LIN {X 0,Y 403.243,Z 462.44,A -85,B 0,C 180,E1 10044.516,E2 10044.516} C_VEL
LIN {X 0,Y 403.34,Z 462.44,A -85,B 0,C 180,E1 10050.792,E2 10050.792} C_VEL
LIN {X 0,Y 403.639,Z 462.44,A -85,B 0,C 180,E1 10057.97,E2 10057.97} C_VEL
LIN {X 0,Y 403.729,Z 462.44,A -85,B 0,C 180,E1 10064.781,E2 10064.781} C_VEL
LIN {X 0,Y 404.101,Z 462.44,A -85,B 0,C 180,E1 10071.38,E2 10071.38} C_VEL
LIN {X 0,Y 404.558,Z 462.44,A -85,B 0,C 180,E1 10077.854,E2 10077.854} C_VEL
LIN {X 0,Y 404.307,Z 462.44,A -85,B 0,C 180,E1 10084.294,E2 10084.294} C_VEL
LIN {X 0,Y 403.998,Z 462.44,A -85,B 0,C 180,E1 10090.798,E2 10090.798} C_VEL
LIN {X 0,Y 403.763,Z 462.44,A -85,B 0,C 180,E1 10097.454,E2 10097.454} C_VEL
LIN {X 0,Y 403.46,Z 462.44,A -85,B 0,C 180,E1 10104.377,E2 10104.377} C_VEL
LIN {X 0,Y 403.325,Z 462.44,A -85,B 0,C 180,E1 10111.701,E2 10111.701} C_VEL
LIN {X 0,Y 403.126,Z 462.44,A -85,B 0,C 180,E1 10117.931,E2 10117.931} C_VEL
LIN {X 0,Y 403.183,Z 462.44,A -85,B 0,C 180,E1 10120.032,E2 10120.032} C_VEL
LIN {X 0,Y 405.626,Z 468.108,A -85,B 0,C 180,E1 10120.64,E2 10120.64} C_VEL
LIN {X 0,Y 425.184,Z 498.302,A -85,B 0,C 180,E1 10124.569,E2 10124.569} C_VEL
LIN {X 0,Y 444.51,Z 533.173,A -85,B 0,C 180,E1 10128.253,E2 10128.253} C_VEL
LIN {X 0,Y 440.339,Z 572.363,A -85,B 0,C 180,E1 10129.774,E2 10129.774} C_VEL
LIN {X 0,Y 434.42,Z 610.186,A -85,B 0,C 180,E1 10132.076,E2 10132.076} C_VEL
LIN {X 0,Y 427.708,Z 644.738,A -85,B 0,C 180,E1 10135.102,E2 10135.102} C_VEL
LIN {X 0,Y 420.828,Z 675.887,A -85,B 0,C 180,E1 10138.855,E2 10138.855} C_VEL
LIN {X 0,Y 414.66,Z 702.51,A -85,B 0,C 180,E1 10143.183,E2 10143.183} C_VEL
LIN {X 0,Y 409.869,Z 724.536,A -85,B 0,C 180,E1 10148.032,E2 10148.032} C_VEL
LIN {X 0,Y 406.864,Z 741.838,A -85,B 0,C 180,E1 10153.237,E2 10153.237} C_VEL
LIN {X 0,Y 405.434,Z 753.406,A -85,B 0,C 180,E1 10158.147,E2 10158.147} C_VEL
LIN {X 0,Y 404.793,Z 761.392,A -85,B 0,C 180,E1 10163.557,E2 10163.557} C_VEL
LIN {X 0,Y 404.608,Z 764.387,A -85,B 0,C 180,E1 10167.855,E2 10167.855} C_VEL
LIN {X 0,Y 404.711,Z 764.342,A -85,B 0,C 180,E1 10172.144,E2 10172.144} C_VEL
LIN {X 0,Y 404.926,Z 759.627,A -85,B 0,C 180,E1 10177.899,E2 10177.899} C_VEL
LIN {X 0,Y 405.887,Z 749.624,A -85,B 0,C 180,E1 10183.577,E2 10183.577} C_VEL
LIN {X 0,Y 407.987,Z 735.102,A -85,B 0,C 180,E1 10188.911,E2 10188.911} C_VEL
LIN {X 0,Y 412.168,Z 713.862,A -85,B 0,C 180,E1 10194.411,E2 10194.411} C_VEL
LIN {X 0,Y 417.696,Z 689.379,A -85,B 0,C 180,E1 10199.022,E2 10199.022} C_VEL
LIN {X 0,Y 424.22,Z 660.818,A -85,B 0,C 180,E1 10203.015,E2 10203.015} C_VEL
LIN {X 0,Y 431.025,Z 628.305,A -85,B 0,C 180,E1 10206.373,E2 10206.373} C_VEL
LIN {X 0,Y 437.479,Z 591.662,A -85,B 0,C 180,E1 10209.075,E2 10209.075} C_VEL
LIN {X 0,Y 442.599,Z 553.853,A -85,B 0,C 180,E1 10210.941,E2 10210.941} C_VEL
LIN {X 0,Y 443.958,Z 532.295,A -85,B 0,C 180,E1 10211.76,E2 10211.76} C_VEL
LIN {X 0,Y 421.037,Z 491.321,A -85,B 0,C 180,E1 10216.122,E2 10216.122} C_VEL
LIN {X 0,Y 405.693,Z 468.193,A -85,B 0,C 180,E1 10219.241,E2 10219.241} C_VEL
LIN {X 0,Y 403.188,Z 463.26,A -85,B 0,C 180,E1 10219.825,E2 10219.825} C_VEL
LIN {X 0,Y 403.085,Z 462.44,A -85,B 0,C 180,E1 10222.077,E2 10222.077} C_VEL
LIN {X 0,Y 403.271,Z 462.44,A -85,B 0,C 180,E1 10228.294,E2 10228.294} C_VEL
LIN {X 0,Y 403.494,Z 462.44,A -85,B 0,C 180,E1 10235.625,E2 10235.625} C_VEL
LIN {X 0,Y 403.856,Z 462.44,A -85,B 0,C 180,E1 10242.55,E2 10242.55} C_VEL
LIN {X 0,Y 404.065,Z 462.44,A -85,B 0,C 180,E1 10249.204,E2 10249.204} C_VEL
LIN {X 0,Y 404.383,Z 462.44,A -85,B 0,C 180,E1 10255.707,E2 10255.707} C_VEL
LIN {X 0,Y 404.56,Z 462.44,A -85,B 0,C 180,E1 10262.146,E2 10262.146} C_VEL
LIN {X 0,Y 404.134,Z 462.44,A -85,B 0,C 180,E1 10268.619,E2 10268.619} C_VEL
LIN {X 0,Y 403.837,Z 462.44,A -85,B 0,C 180,E1 10275.215,E2 10275.215} C_VEL
LIN {X 0,Y 403.621,Z 462.44,A -85,B 0,C 180,E1 10282.031,E2 10282.031} C_VEL
LIN {X 0,Y 403.342,Z 462.44,A -85,B 0,C 180,E1 10289.208,E2 10289.208} C_VEL
LIN {X 0,Y 403.244,Z 462.475,A -85,B 0,C 180,E1 10295.573,E2 10295.573} C_VEL
LIN {X 0,Y 405.552,Z 467.996,A -85,B 0,C 180,E1 10296.151,E2 10296.151} C_VEL
LIN {X 0,Y 424.512,Z 497.638,A -85,B 0,C 180,E1 10300.032,E2 10300.032} C_VEL
LIN {X 0,Y 439.136,Z 526.934,A -85,B 0,C 180,E1 10302.999,E2 10302.999} C_VEL
LIN {X 0,Y 444.863,Z 542.463,A -85,B 0,C 180,E1 10304.377,E2 10304.377} C_VEL
LIN {X 0,Y 439.664,Z 585.502,A -85,B 0,C 180,E1 10306.314,E2 10306.314} C_VEL
LIN {X 0,Y 433.203,Z 625.818,A -85,B 0,C 180,E1 10309.015,E2 10309.015} C_VEL
LIN {X 0,Y 425.789,Z 664.948,A -85,B 0,C 180,E1 10312.666,E2 10312.666} C_VEL
LIN {X 0,Y 418.809,Z 700.533,A -85,B 0,C 180,E1 10317.16,E2 10317.16} C_VEL
LIN {X 0,Y 413.329,Z 728.728,A -85,B 0,C 180,E1 10321.859,E2 10321.859} C_VEL
LIN {X 0,Y 409.238,Z 752.029,A -85,B 0,C 180,E1 10327.011,E2 10327.011} C_VEL
LIN {X 0,Y 408.927,Z 753.833,A -85,B 0,C 180,E1 10327.49,E2 10327.49} C_VEL
LIN {X 0,Y 403.851,Z 761.699,A -85,B 0,C 180,E1 10329.579,E2 10329.579} C_VEL
LIN {X 0,Y 399.002,Z 768.751,A -85,B 0,C 180,E1 10331.769,E2 10331.769} C_VEL
LIN {X 0,Y 397.398,Z 781.94,A -85,B 0,C 180,E1 10337.345,E2 10337.345} C_VEL
LIN {X 0,Y 396.842,Z 790.704,A -85,B 0,C 180,E1 10343.427,E2 10343.427} C_VEL
LIN {X 0,Y 396.811,Z 793.55,A -85,B 0,C 180,E1 10347.813,E2 10347.813} C_VEL
LIN {X 0,Y 396.709,Z 793.546,A -85,B 0,C 180,E1 10352.187,E2 10352.187} C_VEL
LIN {X 0,Y 396.845,Z 789.894,A -85,B 0,C 180,E1 10357.292,E2 10357.292} C_VEL
LIN {X 0,Y 397.495,Z 780.875,A -85,B 0,C 180,E1 10363.212,E2 10363.212} C_VEL
LIN {X 0,Y 399.257,Z 766.259,A -85,B 0,C 180,E1 10369.111,E2 10369.111} C_VEL
LIN {X 0,Y 402.776,Z 744.884,A -85,B 0,C 180,E1 10375.086,E2 10375.086} C_VEL
LIN {X 0,Y 408.167,Z 717.248,A -85,B 0,C 180,E1 10380.668,E2 10380.668} C_VEL
LIN {X 0,Y 415.013,Z 684.684,A -85,B 0,C 180,E1 10385.557,E2 10385.557} C_VEL
LIN {X 0,Y 422.33,Z 649.108,A -85,B 0,C 180,E1 10389.586,E2 10389.586} C_VEL
LIN {X 0,Y 429.644,Z 609.889,A -85,B 0,C 180,E1 10392.846,E2 10392.846} C_VEL
LIN {X 0,Y 436.016,Z 568.538,A -85,B 0,C 180,E1 10395.251,E2 10395.251} C_VEL
LIN {X 0,Y 438.609,Z 543.556,A -85,B 0,C 180,E1 10396.341,E2 10396.341} C_VEL
LIN {X 0,Y 424.38,Z 510.888,A -85,B 0,C 180,E1 10399.602,E2 10399.602} C_VEL
LIN {X 0,Y 405.652,Z 479.832,A -85,B 0,C 180,E1 10403.499,E2 10403.499} C_VEL
LIN {X 0,Y 397.6,Z 467.995,A -85,B 0,C 180,E1 10405.329,E2 10405.329} C_VEL
LIN {X 0,Y 395.292,Z 462.44,A -85,B 0,C 180,E1 10406.071,E2 10406.071} C_VEL
LIN {X 0,Y 395.454,Z 462.44,A -85,B 0,C 180,E1 10412.65,E2 10412.65} C_VEL
LIN {X 0,Y 395.789,Z 462.44,A -85,B 0,C 180,E1 10419.862,E2 10419.862} C_VEL
LIN {X 0,Y 395.862,Z 462.44,A -85,B 0,C 180,E1 10426.733,E2 10426.733} C_VEL
LIN {X 0,Y 396.337,Z 462.44,A -85,B 0,C 180,E1 10433.418,E2 10433.418} C_VEL
LIN {X 0,Y 396.597,Z 462.44,A -85,B 0,C 180,E1 10439.999,E2 10439.999} C_VEL
LIN {X 0,Y 396.285,Z 462.44,A -85,B 0,C 180,E1 10446.58,E2 10446.58} C_VEL
LIN {X 0,Y 395.984,Z 462.44,A -85,B 0,C 180,E1 10453.26,E2 10453.26} C_VEL
LIN {X 0,Y 395.741,Z 462.44,A -85,B 0,C 180,E1 10460.138,E2 10460.138} C_VEL
LIN {X 0,Y 395.426,Z 462.44,A -85,B 0,C 180,E1 10467.35,E2 10467.35} C_VEL
LIN {X 0,Y 395.339,Z 462.44,A -85,B 0,C 180,E1 10472.585,E2 10472.585} C_VEL
LIN {X 0,Y 395.199,Z 462.44,A -85,B 0,C 180,E1 10478.508,E2 10478.508} C_VEL
LIN {X 0,Y 397.442,Z 467.939,A -85,B 0,C 180,E1 10479.116,E2 10479.116} C_VEL
LIN {X 0,Y 405.055,Z 478.925,A -85,B 0,C 180,E1 10480.822,E2 10480.822} C_VEL
LIN {X 0,Y 425.307,Z 511.342,A -85,B 0,C 180,E1 10484.919,E2 10484.919} C_VEL
LIN {X 0,Y 438.604,Z 537.518,A -85,B 0,C 180,E1 10487.683,E2 10487.683} C_VEL
LIN {X 0,Y 434.209,Z 574.487,A -85,B 0,C 180,E1 10489.169,E2 10489.169} C_VEL
LIN {X 0,Y 428.051,Z 611.767,A -85,B 0,C 180,E1 10491.495,E2 10491.495} C_VEL
LIN {X 0,Y 421.059,Z 645.965,A -85,B 0,C 180,E1 10494.552,E2 10494.552} C_VEL
LIN {X 0,Y 413.986,Z 676.406,A -85,B 0,C 180,E1 10498.281,E2 10498.281} C_VEL
LIN {X 0,Y 407.423,Z 703.332,A -85,B 0,C 180,E1 10502.736,E2 10502.736} C_VEL
LIN {X 0,Y 402.422,Z 725.088,A -85,B 0,C 180,E1 10507.603,E2 10507.603} C_VEL
LIN {X 0,Y 399.181,Z 742.302,A -85,B 0,C 180,E1 10512.905,E2 10512.905} C_VEL
LIN {X 0,Y 397.628,Z 753.785,A -85,B 0,C 180,E1 10517.911,E2 10517.911} C_VEL
LIN {X 0,Y 396.907,Z 761.705,A -85,B 0,C 180,E1 10523.428,E2 10523.428} C_VEL
LIN {X 0,Y 396.71,Z 764.677,A -85,B 0,C 180,E1 10527.813,E2 10527.813} C_VEL
LIN {X 0,Y 396.811,Z 764.633,A -85,B 0,C 180,E1 10532.187,E2 10532.187} C_VEL
LIN {X 0,Y 397.004,Z 760.642,A -85,B 0,C 180,E1 10537.487,E2 10537.487} C_VEL
LIN {X 0,Y 397.944,Z 751.414,A -85,B 0,C 180,E1 10543.197,E2 10543.197} C_VEL
LIN {X 0,Y 400.43,Z 735.516,A -85,B 0,C 180,E1 10549.319,E2 10549.319} C_VEL
LIN {X 0,Y 404.835,Z 714.398,A -85,B 0,C 180,E1 10554.883,E2 10554.883} C_VEL
LIN {X 0,Y 410.779,Z 689.583,A -85,B 0,C 180,E1 10559.617,E2 10559.617} C_VEL
LIN {X 0,Y 417.86,Z 659.909,A -85,B 0,C 180,E1 10563.79,E2 10563.79} C_VEL
LIN {X 0,Y 424.831,Z 628.177,A -85,B 0,C 180,E1 10567.074,E2 10567.074} C_VEL
LIN {X 0,Y 431.426,Z 592.294,A -85,B 0,C 180,E1 10569.748,E2 10569.748} C_VEL
LIN {X 0,Y 436.852,Z 554.113,A -85,B 0,C 180,E1 10571.648,E2 10571.648} C_VEL
LIN {X 0,Y 438.104,Z 535.545,A -85,B 0,C 180,E1 10572.372,E2 10572.372} C_VEL
LIN {X 0,Y 417.025,Z 497.141,A -85,B 0,C 180,E1 10576.609,E2 10576.609} C_VEL
LIN {X 0,Y 398.095,Z 468.555,A -85,B 0,C 180,E1 10580.634,E2 10580.634} C_VEL
LIN {X 0,Y 395.27,Z 463.755,A -85,B 0,C 180,E1 10581.317,E2 10581.317} C_VEL
LIN {X 0,Y 395.179,Z 462.44,A -85,B 0,C 180,E1 10581.434,E2 10581.434} C_VEL
LIN {X 0,Y 395.269,Z 462.44,A -85,B 0,C 180,E1 10587.574,E2 10587.574} C_VEL
LIN {X 0,Y 395.439,Z 462.44,A -85,B 0,C 180,E1 10592.651,E2 10592.651} C_VEL
LIN {X 0,Y 395.796,Z 462.44,A -85,B 0,C 180,E1 10599.865,E2 10599.865} C_VEL
LIN {X 0,Y 396.074,Z 462.44,A -85,B 0,C 180,E1 10606.743,E2 10606.743} C_VEL
LIN {X 0,Y 396.308,Z 462.44,A -85,B 0,C 180,E1 10613.42,E2 10613.42} C_VEL
LIN {X 0,Y 396.666,Z 462.44,A -85,B 0,C 180,E1 10620.001,E2 10620.001} C_VEL
LIN {X 0,Y 396.332,Z 462.44,A -85,B 0,C 180,E1 10626.637,E2 10626.637} C_VEL
LIN {X 0,Y 395.991,Z 462.44,A -85,B 0,C 180,E1 10633.263,E2 10633.263} C_VEL
LIN {X 0,Y 395.757,Z 462.44,A -85,B 0,C 180,E1 10640.14,E2 10640.14} C_VEL
LIN {X 0,Y 395.457,Z 462.44,A -85,B 0,C 180,E1 10647.35,E2 10647.35} C_VEL
LIN {X 0,Y 395.333,Z 462.763,A -85,B 0,C 180,E1 10654.086,E2 10654.086} C_VEL
LIN {X 0,Y 397.8,Z 468.188,A -85,B 0,C 180,E1 10654.732,E2 10654.732} C_VEL
LIN {X 0,Y 414.691,Z 494.071,A -85,B 0,C 180,E1 10658.429,E2 10658.429} C_VEL
LIN {X 0,Y 430.735,Z 523.96,A -85,B 0,C 180,E1 10661.779,E2 10661.779} C_VEL
LIN {X 0,Y 438.795,Z 545.274,A -85,B 0,C 180,E1 10663.776,E2 10663.776} C_VEL
LIN {X 0,Y 433.486,Z 586.598,A -85,B 0,C 180,E1 10665.686,E2 10665.686} C_VEL
LIN {X 0,Y 426.751,Z 626.42,A -85,B 0,C 180,E1 10668.397,E2 10668.397} C_VEL
LIN {X 0,Y 419.033,Z 665.305,A -85,B 0,C 180,E1 10672.1,E2 10672.1} C_VEL
LIN {X 0,Y 411.788,Z 699.678,A -85,B 0,C 180,E1 10676.527,E2 10676.527} C_VEL
LIN {X 0,Y 405.725,Z 729.414,A -85,B 0,C 180,E1 10681.587,E2 10681.587} C_VEL
LIN {X 0,Y 401.316,Z 753.319,A -85,B 0,C 180,E1 10687.039,E2 10687.039} C_VEL
LIN {X 0,Y 399.002,Z 768.751,A -85,B 0,C 180,E1 10691.769,E2 10691.769} C_VEL
LIN {X 0,Y 395.882,Z 773.516,A -85,B 0,C 180,E1 10693.479,E2 10693.479} C_VEL
LIN {X 0,Y 389.845,Z 779.624,A -85,B 0,C 180,E1 10696.09,E2 10696.09} C_VEL
LIN {X 0,Y 389.698,Z 780.266,A -85,B 0,C 180,E1 10696.398,E2 10696.398} C_VEL
LIN {X 0,Y 388.936,Z 789.6,A -85,B 0,C 180,E1 10702.571,E2 10702.571} C_VEL
LIN {X 0,Y 388.915,Z 793.26,A -85,B 0,C 180,E1 10707.769,E2 10707.769} C_VEL
LIN {X 0,Y 388.82,Z 793.257,A -85,B 0,C 180,E1 10712.232,E2 10712.232} C_VEL
LIN {X 0,Y 388.951,Z 789.583,A -85,B 0,C 180,E1 10717.441,E2 10717.441} C_VEL
LIN {X 0,Y 389.639,Z 780.512,A -85,B 0,C 180,E1 10723.483,E2 10723.483} C_VEL
LIN {X 0,Y 391.56,Z 765.572,A -85,B 0,C 180,E1 10729.588,E2 10729.588} C_VEL
LIN {X 0,Y 395.241,Z 744.563,A -85,B 0,C 180,E1 10735.522,E2 10735.522} C_VEL
LIN {X 0,Y 400.986,Z 716.49,A -85,B 0,C 180,E1 10741.279,E2 10741.279} C_VEL
LIN {X 0,Y 408.135,Z 684.775,A -85,B 0,C 180,E1 10746.143,E2 10746.143} C_VEL
LIN {X 0,Y 415.777,Z 649.522,A -85,B 0,C 180,E1 10750.208,E2 10750.208} C_VEL
LIN {X 0,Y 423.285,Z 611.364,A -85,B 0,C 180,E1 10753.443,E2 10753.443} C_VEL
LIN {X 0,Y 430.124,Z 569.177,A -85,B 0,C 180,E1 10755.939,E2 10755.939} C_VEL
LIN {X 0,Y 432.454,Z 546.358,A -85,B 0,C 180,E1 10756.977,E2 10756.977} C_VEL
LIN {X 0,Y 419.8,Z 516.142,A -85,B 0,C 180,E1 10760.099,E2 10760.099} C_VEL
LIN {X 0,Y 401.79,Z 485.729,A -85,B 0,C 180,E1 10764.013,E2 10764.013} C_VEL
LIN {X 0,Y 389.978,Z 468.304,A -85,B 0,C 180,E1 10766.833,E2 10766.833} C_VEL
LIN {X 0,Y 387.541,Z 463.879,A -85,B 0,C 180,E1 10767.49,E2 10767.49} C_VEL
LIN {X 0,Y 387.379,Z 462.44,A -85,B 0,C 180,E1 10767.797,E2 10767.797} C_VEL
LIN {X 0,Y 387.575,Z 462.44,A -85,B 0,C 180,E1 10774.551,E2 10774.551} C_VEL
LIN {X 0,Y 387.855,Z 462.44,A -85,B 0,C 180,E1 10781.803,E2 10781.803} C_VEL
LIN {X 0,Y 388.016,Z 462.44,A -85,B 0,C 180,E1 10788.749,E2 10788.749} C_VEL
LIN {X 0,Y 388.477,Z 462.44,A -85,B 0,C 180,E1 10795.528,E2 10795.528} C_VEL
LIN {X 0,Y 388.705,Z 462.44,A -85,B 0,C 180,E1 10799.999,E2 10799.999} C_VEL
LIN {X 0,Y 388.362,Z 462.44,A -85,B 0,C 180,E1 10806.715,E2 10806.715} C_VEL
LIN {X 0,Y 388.056,Z 462.44,A -85,B 0,C 180,E1 10813.536,E2 10813.536} C_VEL
LIN {X 0,Y 387.764,Z 462.44,A -85,B 0,C 180,E1 10820.571,E2 10820.571} C_VEL
LIN {X 0,Y 387.523,Z 462.44,A -85,B 0,C 180,E1 10827.956,E2 10827.956} C_VEL
LIN {X 0,Y 387.352,Z 462.44,A -85,B 0,C 180,E1 10835.891,E2 10835.891} C_VEL
LIN {X 0,Y 387.335,Z 462.608,A -85,B 0,C 180,E1 10836.907,E2 10836.907} C_VEL
LIN {X 0,Y 389.422,Z 467.801,A -85,B 0,C 180,E1 10837.505,E2 10837.505} C_VEL
LIN {X 0,Y 392.445,Z 471.944,A -85,B 0,C 180,E1 10838.246,E2 10838.246} C_VEL
LIN {X 0,Y 408.063,Z 495.276,A -85,B 0,C 180,E1 10841.77,E2 10841.77} C_VEL
LIN {X 0,Y 427.465,Z 529.122,A -85,B 0,C 180,E1 10845.822,E2 10845.822} C_VEL
LIN {X 0,Y 432.724,Z 539.783,A -85,B 0,C 180,E1 10847.006,E2 10847.006} C_VEL
LIN {X 0,Y 427.988,Z 577.783,A -85,B 0,C 180,E1 10848.614,E2 10848.614} C_VEL
LIN {X 0,Y 421.648,Z 613.614,A -85,B 0,C 180,E1 10850.916,E2 10850.916} C_VEL
LIN {X 0,Y 414.438,Z 647.187,A -85,B 0,C 180,E1 10853.986,E2 10853.986} C_VEL
LIN {X 0,Y 407.189,Z 676.889,A -85,B 0,C 180,E1 10857.688,E2 10857.688} C_VEL
LIN {X 0,Y 400.448,Z 703.232,A -85,B 0,C 180,E1 10862.101,E2 10862.101} C_VEL
LIN {X 0,Y 395.121,Z 725.015,A -85,B 0,C 180,E1 10867.019,E2 10867.019} C_VEL
LIN {X 0,Y 391.537,Z 742.753,A -85,B 0,C 180,E1 10872.56,E2 10872.56} C_VEL
LIN {X 0,Y 389.833,Z 754.166,A -85,B 0,C 180,E1 10877.665,E2 10877.665} C_VEL
LIN {X 0,Y 389.041,Z 762.018,A -85,B 0,C 180,E1 10883.295,E2 10883.295} C_VEL
LIN {X 0,Y 388.821,Z 764.968,A -85,B 0,C 180,E1 10887.768,E2 10887.768} C_VEL
LIN {X 0,Y 388.914,Z 764.925,A -85,B 0,C 180,E1 10892.231,E2 10892.231} C_VEL
LIN {X 0,Y 389.125,Z 760.966,A -85,B 0,C 180,E1 10897.64,E2 10897.64} C_VEL
LIN {X 0,Y 390.152,Z 751.813,A -85,B 0,C 180,E1 10903.465,E2 10903.465} C_VEL
LIN {X 0,Y 392.641,Z 737.037,A -85,B 0,C 180,E1 10909.357,E2 10909.357} C_VEL
LIN {X 0,Y 397.259,Z 716.128,A -85,B 0,C 180,E1 10915.089,E2 10915.089} C_VEL
LIN {X 0,Y 403.73,Z 690.395,A -85,B 0,C 180,E1 10920.126,E2 10920.126} C_VEL
LIN {X 0,Y 411.219,Z 660.619,A -85,B 0,C 180,E1 10924.387,E2 10924.387} C_VEL
LIN {X 0,Y 418.595,Z 628.581,A -85,B 0,C 180,E1 10927.747,E2 10927.747} C_VEL
LIN {X 0,Y 425.592,Z 592.054,A -85,B 0,C 180,E1 10930.488,E2 10930.488} C_VEL
LIN {X 0,Y 431.171,Z 554.253,A -85,B 0,C 180,E1 10932.379,E2 10932.379} C_VEL
LIN {X 0,Y 432.208,Z 538.753,A -85,B 0,C 180,E1 10933.013,E2 10933.013} C_VEL
LIN {X 0,Y 412.626,Z 502.339,A -85,B 0,C 180,E1 10937.189,E2 10937.189} C_VEL
LIN {X 0,Y 394.373,Z 474.672,A -85,B 0,C 180,E1 10941.184,E2 10941.184} C_VEL
LIN {X 0,Y 389.32,Z 467.696,A -85,B 0,C 180,E1 10942.409,E2 10942.409} C_VEL
LIN {X 0,Y 387.274,Z 462.44,A -85,B 0,C 180,E1 10943.056,E2 10943.056} C_VEL
LIN {X 0,Y 387.385,Z 462.44,A -85,B 0,C 180,E1 10949.467,E2 10949.467} C_VEL
LIN {X 0,Y 387.694,Z 462.44,A -85,B 0,C 180,E1 10957.016,E2 10957.016} C_VEL
LIN {X 0,Y 388.062,Z 462.44,A -85,B 0,C 180,E1 10964.153,E2 10964.153} C_VEL
LIN {X 0,Y 388.281,Z 462.44,A -85,B 0,C 180,E1 10971.269,E2 10971.269} C_VEL
LIN {X 0,Y 388.681,Z 462.44,A -85,B 0,C 180,E1 10977.769,E2 10977.769} C_VEL
LIN {X 0,Y 388.48,Z 462.44,A -85,B 0,C 180,E1 10984.472,E2 10984.472} C_VEL
LIN {X 0,Y 388.121,Z 462.44,A -85,B 0,C 180,E1 10991.248,E2 10991.248} C_VEL
LIN {X 0,Y 387.863,Z 462.44,A -85,B 0,C 180,E1 10998.197,E2 10998.197} C_VEL
LIN {X 0,Y 387.577,Z 462.44,A -85,B 0,C 180,E1 11005.449,E2 11005.449} C_VEL
LIN {X 0,Y 387.407,Z 462.44,A -85,B 0,C 180,E1 11012.442,E2 11012.442} C_VEL
LIN {X 0,Y 389.657,Z 467.996,A -85,B 0,C 180,E1 11013.109,E2 11013.109} C_VEL
LIN {X 0,Y 392.574,Z 472.095,A -85,B 0,C 180,E1 11013.835,E2 11013.835} C_VEL
LIN {X 0,Y 409.993,Z 498.604,A -85,B 0,C 180,E1 11017.79,E2 11017.79} C_VEL
LIN {X 0,Y 425.494,Z 528.178,A -85,B 0,C 180,E1 11021.212,E2 11021.212} C_VEL
LIN {X 0,Y 432.694,Z 548.803,A -85,B 0,C 180,E1 11023.191,E2 11023.191} C_VEL
LIN {X 0,Y 427.359,Z 587.739,A -85,B 0,C 180,E1 11025.044,E2 11025.044} C_VEL
LIN {X 0,Y 420.354,Z 627.093,A -85,B 0,C 180,E1 11027.769,E2 11027.769} C_VEL
LIN {X 0,Y 412.507,Z 664.691,A -85,B 0,C 180,E1 11031.391,E2 11031.391} C_VEL
LIN {X 0,Y 404.825,Z 699.054,A -85,B 0,C 180,E1 11035.873,E2 11035.873} C_VEL
LIN {X 0,Y 398.384,Z 728.808,A -85,B 0,C 180,E1 11041.039,E2 11041.039} C_VEL
LIN {X 0,Y 393.818,Z 752.47,A -85,B 0,C 180,E1 11046.491,E2 11046.491} C_VEL
LIN {X 0,Y 390.779,Z 771.449,A -85,B 0,C 180,E1 11052.525,E2 11052.525} C_VEL
LIN {X 0,Y 389.698,Z 780.266,A -85,B 0,C 180,E1 11056.398,E2 11056.398} C_VEL
LIN {X 0,Y 386.9,Z 783.741,A -85,B 0,C 180,E1 11058.22,E2 11058.22} C_VEL
LIN {X 0,Y 381.229,Z 787.741,A -85,B 0,C 180,E1 11061.005,E2 11061.005} C_VEL
LIN {X 0,Y 381.102,Z 788.082,A -85,B 0,C 180,E1 11061.332,E2 11061.332} C_VEL
LIN {X 0,Y 380.951,Z 791.891,A -85,B 0,C 180,E1 11065.441,E2 11065.441} C_VEL
LIN {X 0,Y 381.01,Z 793.329,A -85,B 0,C 180,E1 11070,E2 11070} C_VEL
LIN {X 0,Y 380.927,Z 791.891,A -85,B 0,C 180,E1 11074.56,E2 11074.56} C_VEL
LIN {X 0,Y 381.299,Z 785.926,A -85,B 0,C 180,E1 11080.294,E2 11080.294} C_VEL
LIN {X 0,Y 382.408,Z 775.209,A -85,B 0,C 180,E1 11086.091,E2 11086.091} C_VEL
LIN {X 0,Y 385.045,Z 758.047,A -85,B 0,C 180,E1 11092.242,E2 11092.242} C_VEL
LIN {X 0,Y 389.739,Z 734.384,A -85,B 0,C 180,E1 11098.249,E2 11098.249} C_VEL
LIN {X 0,Y 396.366,Z 705.806,A -85,B 0,C 180,E1 11103.635,E2 11103.635} C_VEL
LIN {X 0,Y 403.963,Z 673.635,A -85,B 0,C 180,E1 11108.205,E2 11108.205} C_VEL
LIN {X 0,Y 412.054,Z 637.549,A -85,B 0,C 180,E1 11112.028,E2 11112.028} C_VEL
LIN {X 0,Y 419.82,Z 597.766,A -85,B 0,C 180,E1 11115.077,E2 11115.077} C_VEL
LIN {X 0,Y 426.104,Z 556.005,A -85,B 0,C 180,E1 11117.286,E2 11117.286} C_VEL
LIN {X 0,Y 426.333,Z 548.846,A -85,B 0,C 180,E1 11117.653,E2 11117.653} C_VEL
LIN {X 0,Y 414.639,Z 520.428,A -85,B 0,C 180,E1 11120.714,E2 11120.714} C_VEL
LIN {X 0,Y 397.507,Z 490.866,A -85,B 0,C 180,E1 11124.646,E2 11124.646} C_VEL
LIN {X 0,Y 382.488,Z 468.624,A -85,B 0,C 180,E1 11128.429,E2 11128.429} C_VEL
LIN {X 0,Y 379.581,Z 463.619,A -85,B 0,C 180,E1 11129.267,E2 11129.267} C_VEL
LIN {X 0,Y 379.525,Z 462.44,A -85,B 0,C 180,E1 11129.428,E2 11129.428} C_VEL
LIN {X 0,Y 379.739,Z 462.44,A -85,B 0,C 180,E1 11136.503,E2 11136.503} C_VEL
LIN {X 0,Y 379.949,Z 462.44,A -85,B 0,C 180,E1 11143.803,E2 11143.803} C_VEL
LIN {X 0,Y 380.3,Z 462.44,A -85,B 0,C 180,E1 11150.836,E2 11150.836} C_VEL
LIN {X 0,Y 380.833,Z 462.44,A -85,B 0,C 180,E1 11157.72,E2 11157.72} C_VEL
LIN {X 0,Y 380.571,Z 462.44,A -85,B 0,C 180,E1 11164.562,E2 11164.562} C_VEL
LIN {X 0,Y 380.2,Z 462.44,A -85,B 0,C 180,E1 11171.483,E2 11171.483} C_VEL
LIN {X 0,Y 379.922,Z 462.44,A -85,B 0,C 180,E1 11178.589,E2 11178.589} C_VEL
LIN {X 0,Y 379.626,Z 462.44,A -85,B 0,C 180,E1 11186.018,E2 11186.018} C_VEL
LIN {X 0,Y 379.443,Z 462.44,A -85,B 0,C 180,E1 11193.957,E2 11193.957} C_VEL
LIN {X 0,Y 379.502,Z 463.265,A -85,B 0,C 180,E1 11195.176,E2 11195.176} C_VEL
LIN {X 0,Y 382.246,Z 468.462,A -85,B 0,C 180,E1 11195.972,E2 11195.972} C_VEL
LIN {X 0,Y 397.826,Z 491.087,A -85,B 0,C 180,E1 11199.829,E2 11199.829} C_VEL
LIN {X 0,Y 417.024,Z 523.235,A -85,B 0,C 180,E1 11204.061,E2 11204.061} C_VEL
LIN {X 0,Y 426.858,Z 543.914,A -85,B 0,C 180,E1 11206.388,E2 11206.388} C_VEL
LIN {X 0,Y 421.449,Z 583.428,A -85,B 0,C 180,E1 11208.172,E2 11208.172} C_VEL
LIN {X 0,Y 414.23,Z 620.638,A -85,B 0,C 180,E1 11210.735,E2 11210.735} C_VEL
LIN {X 0,Y 406.113,Z 655.513,A -85,B 0,C 180,E1 11214.205,E2 11214.205} C_VEL
LIN {X 0,Y 398.416,Z 684.842,A -85,B 0,C 180,E1 11218.21,E2 11218.21} C_VEL
LIN {X 0,Y 391.508,Z 710.43,A -85,B 0,C 180,E1 11222.943,E2 11222.943} C_VEL
LIN {X 0,Y 386.391,Z 731.07,A -85,B 0,C 180,E1 11228.144,E2 11228.144} C_VEL
LIN {X 0,Y 383.093,Z 747.449,A -85,B 0,C 180,E1 11233.939,E2 11233.939} C_VEL
LIN {X 0,Y 381.598,Z 758.283,A -85,B 0,C 180,E1 11239.714,E2 11239.714} C_VEL
LIN {X 0,Y 380.961,Z 764.161,A -85,B 0,C 180,E1 11245.441,E2 11245.441} C_VEL
LIN {X 0,Y 381.01,Z 765.618,A -85,B 0,C 180,E1 11250,E2 11250} C_VEL
LIN {X 0,Y 380.978,Z 764.097,A -85,B 0,C 180,E1 11254.559,E2 11254.559} C_VEL
LIN {X 0,Y 381.612,Z 758.146,A -85,B 0,C 180,E1 11260.285,E2 11260.285} C_VEL
LIN {X 0,Y 383.107,Z 747.252,A -85,B 0,C 180,E1 11266.061,E2 11266.061} C_VEL
LIN {X 0,Y 386.707,Z 729.786,A -85,B 0,C 180,E1 11272.14,E2 11272.14} C_VEL
LIN {X 0,Y 392.328,Z 707.456,A -85,B 0,C 180,E1 11277.589,E2 11277.589} C_VEL
LIN {X 0,Y 399.586,Z 680.53,A -85,B 0,C 180,E1 11282.36,E2 11282.36} C_VEL
LIN {X 0,Y 407.429,Z 650.088,A -85,B 0,C 180,E1 11286.319,E2 11286.319} C_VEL
LIN {X 0,Y 415.129,Z 616.507,A -85,B 0,C 180,E1 11289.494,E2 11289.494} C_VEL
LIN {X 0,Y 421.745,Z 580.922,A -85,B 0,C 180,E1 11291.878,E2 11291.878} C_VEL
LIN {X 0,Y 426.484,Z 542.229,A -85,B 0,C 180,E1 11293.643,E2 11293.643} C_VEL
LIN {X 0,Y 407.388,Z 506.122,A -85,B 0,C 180,E1 11297.956,E2 11297.956} C_VEL
LIN {X 0,Y 390.546,Z 480.485,A -85,B 0,C 180,E1 11301.781,E2 11301.781} C_VEL
LIN {X 0,Y 382.29,Z 468.546,A -85,B 0,C 180,E1 11303.903,E2 11303.903} C_VEL
LIN {X 0,Y 379.426,Z 463.324,A -85,B 0,C 180,E1 11304.724,E2 11304.724} C_VEL
LIN {X 0,Y 379.42,Z 462.44,A -85,B 0,C 180,E1 11305.2,E2 11305.2} C_VEL
LIN {X 0,Y 379.529,Z 462.44,A -85,B 0,C 180,E1 11311.402,E2 11311.402} C_VEL
LIN {X 0,Y 379.851,Z 462.44,A -85,B 0,C 180,E1 11318.98,E2 11318.98} C_VEL
LIN {X 0,Y 380.187,Z 462.44,A -85,B 0,C 180,E1 11326.178,E2 11326.178} C_VEL
LIN {X 0,Y 380.489,Z 462.44,A -85,B 0,C 180,E1 11333.146,E2 11333.146} C_VEL
LIN {X 0,Y 380.869,Z 462.44,A -85,B 0,C 180,E1 11340.001,E2 11340.001} C_VEL
LIN {X 0,Y 380.536,Z 462.44,A -85,B 0,C 180,E1 11346.856,E2 11346.856} C_VEL
LIN {X 0,Y 380.116,Z 462.44,A -85,B 0,C 180,E1 11353.827,E2 11353.827} C_VEL
LIN {X 0,Y 379.841,Z 462.44,A -85,B 0,C 180,E1 11361.023,E2 11361.023} C_VEL
LIN {X 0,Y 379.547,Z 462.44,A -85,B 0,C 180,E1 11368.64,E2 11368.64} C_VEL
LIN {X 0,Y 379.55,Z 463.245,A -85,B 0,C 180,E1 11370.736,E2 11370.736} C_VEL
LIN {X 0,Y 382.238,Z 468.448,A -85,B 0,C 180,E1 11371.532,E2 11371.532} C_VEL
LIN {X 0,Y 396.752,Z 489.652,A -85,B 0,C 180,E1 11375.192,E2 11375.192} C_VEL
LIN {X 0,Y 414.36,Z 519.858,A -85,B 0,C 180,E1 11379.229,E2 11379.229} C_VEL
LIN {X 0,Y 425.95,Z 547.76,A -85,B 0,C 180,E1 11382.24,E2 11382.24} C_VEL
LIN {X 0,Y 426.529,Z 552.791,A -85,B 0,C 180,E1 11382.598,E2 11382.598} C_VEL
LIN {X 0,Y 420.808,Z 591.846,A -85,B 0,C 180,E1 11384.564,E2 11384.564} C_VEL
LIN {X 0,Y 413.84,Z 628.638,A -85,B 0,C 180,E1 11387.195,E2 11387.195} C_VEL
LIN {X 0,Y 405.689,Z 665.745,A -85,B 0,C 180,E1 11390.854,E2 11390.854} C_VEL
LIN {X 0,Y 397.99,Z 698.52,A -85,B 0,C 180,E1 11395.203,E2 11395.203} C_VEL
LIN {X 0,Y 391.14,Z 728.204,A -85,B 0,C 180,E1 11400.45,E2 11400.45} C_VEL
LIN {X 0,Y 386.04,Z 752.939,A -85,B 0,C 180,E1 11406.295,E2 11406.295} C_VEL
LIN {X 0,Y 383.048,Z 771.011,A -85,B 0,C 180,E1 11412.161,E2 11412.161} C_VEL
LIN {X 0,Y 381.39,Z 784.243,A -85,B 0,C 180,E1 11418.551,E2 11418.551} C_VEL
LIN {X 0,Y 381.102,Z 788.082,A -85,B 0,C 180,E1 11421.332,E2 11421.332} C_VEL
LIN {X 0,Y 378.45,Z 790.116,A -85,B 0,C 180,E1 11423.243,E2 11423.243} C_VEL
LIN {X 0,Y 373.102,Z 791.981,A -85,B 0,C 180,E1 11426.138,E2 11426.138} C_VEL
LIN {X 0,Y 373.013,Z 792.122,A -85,B 0,C 180,E1 11426.475,E2 11426.475} C_VEL
LIN {X 0,Y 373.138,Z 793.043,A -85,B 0,C 180,E1 11430,E2 11430} C_VEL
LIN {X 0,Y 373.052,Z 791.595,A -85,B 0,C 180,E1 11434.656,E2 11434.656} C_VEL
LIN {X 0,Y 373.421,Z 785.585,A -85,B 0,C 180,E1 11440.513,E2 11440.513} C_VEL
LIN {X 0,Y 374.604,Z 774.789,A -85,B 0,C 180,E1 11446.436,E2 11446.436} C_VEL
LIN {X 0,Y 377.445,Z 757.567,A -85,B 0,C 180,E1 11452.696,E2 11452.696} C_VEL
LIN {X 0,Y 382.325,Z 734.436,A -85,B 0,C 180,E1 11458.718,E2 11458.718} C_VEL
LIN {X 0,Y 389.406,Z 705.3,A -85,B 0,C 180,E1 11464.319,E2 11464.319} C_VEL
LIN {X 0,Y 397.527,Z 673.117,A -85,B 0,C 180,E1 11468.935,E2 11468.935} C_VEL
LIN {X 0,Y 405.999,Z 636.88,A -85,B 0,C 180,E1 11472.807,E2 11472.807} C_VEL
LIN {X 0,Y 413.953,Z 597.847,A -85,B 0,C 180,E1 11475.821,E2 11475.821} C_VEL
LIN {X 0,Y 420.609,Z 555.138,A -85,B 0,C 180,E1 11478.085,E2 11478.085} C_VEL
LIN {X 0,Y 419.345,Z 548.587,A -85,B 0,C 180,E1 11478.64,E2 11478.64} C_VEL
LIN {X 0,Y 407.727,Z 521.035,A -85,B 0,C 180,E1 11481.794,E2 11481.794} C_VEL
LIN {X 0,Y 390.692,Z 492.079,A -85,B 0,C 180,E1 11485.923,E2 11485.923} C_VEL
LIN {X 0,Y 378.223,Z 474.046,A -85,B 0,C 180,E1 11489.212,E2 11489.212} C_VEL
LIN {X 0,Y 374.692,Z 468.726,A -85,B 0,C 180,E1 11490.248,E2 11490.248} C_VEL
LIN {X 0,Y 371.735,Z 463.859,A -85,B 0,C 180,E1 11491.168,E2 11491.168} C_VEL
LIN {X 0,Y 371.633,Z 462.44,A -85,B 0,C 180,E1 11491.414,E2 11491.414} C_VEL
LIN {X 0,Y 371.879,Z 462.44,A -85,B 0,C 180,E1 11498.505,E2 11498.505} C_VEL
LIN {X 0,Y 372.069,Z 462.44,A -85,B 0,C 180,E1 11505.868,E2 11505.868} C_VEL
LIN {X 0,Y 372.595,Z 462.44,A -85,B 0,C 180,E1 11512.997,E2 11512.997} C_VEL
LIN {X 0,Y 372.902,Z 462.44,A -85,B 0,C 180,E1 11519.999,E2 11519.999} C_VEL
LIN {X 0,Y 372.524,Z 462.44,A -85,B 0,C 180,E1 11527.002,E2 11527.002} C_VEL
LIN {X 0,Y 372.165,Z 462.44,A -85,B 0,C 180,E1 11534.126,E2 11534.126} C_VEL
LIN {X 0,Y 371.826,Z 462.44,A -85,B 0,C 180,E1 11541.495,E2 11541.495} C_VEL
LIN {X 0,Y 371.639,Z 462.44,A -85,B 0,C 180,E1 11546.621,E2 11546.621} C_VEL
LIN {X 0,Y 371.576,Z 462.686,A -85,B 0,C 180,E1 11553.216,E2 11553.216} C_VEL
LIN {X 0,Y 373.707,Z 467.84,A -85,B 0,C 180,E1 11553.933,E2 11553.933} C_VEL
LIN {X 0,Y 376.458,Z 470.959,A -85,B 0,C 180,E1 11554.708,E2 11554.708} C_VEL
LIN {X 0,Y 396.245,Z 500.094,A -85,B 0,C 180,E1 11559.779,E2 11559.779} C_VEL
LIN {X 0,Y 414.948,Z 533.455,A -85,B 0,C 180,E1 11564.156,E2 11564.156} C_VEL
LIN {X 0,Y 420.993,Z 547.013,A -85,B 0,C 180,E1 11565.725,E2 11565.725} C_VEL
LIN {X 0,Y 415.416,Z 585.253,A -85,B 0,C 180,E1 11567.512,E2 11567.512} C_VEL
LIN {X 0,Y 407.818,Z 622.525,A -85,B 0,C 180,E1 11570.145,E2 11570.145} C_VEL
LIN {X 0,Y 399.662,Z 655.996,A -85,B 0,C 180,E1 11573.535,E2 11573.535} C_VEL
LIN {X 0,Y 391.433,Z 685.898,A -85,B 0,C 180,E1 11577.696,E2 11577.696} C_VEL
LIN {X 0,Y 384.323,Z 710.821,A -85,B 0,C 180,E1 11582.395,E2 11582.395} C_VEL
LIN {X 0,Y 378.886,Z 731.437,A -85,B 0,C 180,E1 11587.688,E2 11587.688} C_VEL
LIN {X 0,Y 375.378,Z 747.794,A -85,B 0,C 180,E1 11593.599,E2 11593.599} C_VEL
LIN {X 0,Y 373.748,Z 758.61,A -85,B 0,C 180,E1 11599.496,E2 11599.496} C_VEL
LIN {X 0,Y 373.088,Z 764.461,A -85,B 0,C 180,E1 11605.344,E2 11605.344} C_VEL
LIN {X 0,Y 373.137,Z 765.904,A -85,B 0,C 180,E1 11610,E2 11610} C_VEL
LIN {X 0,Y 373.104,Z 764.396,A -85,B 0,C 180,E1 11614.656,E2 11614.656} C_VEL
LIN {X 0,Y 373.762,Z 758.479,A -85,B 0,C 180,E1 11620.504,E2 11620.504} C_VEL
LIN {X 0,Y 375.399,Z 747.599,A -85,B 0,C 180,E1 11626.4,E2 11626.4} C_VEL
LIN {X 0,Y 379.246,Z 730.167,A -85,B 0,C 180,E1 11632.599,E2 11632.599} C_VEL
LIN {X 0,Y 385.201,Z 707.866,A -85,B 0,C 180,E1 11638.144,E2 11638.144} C_VEL
LIN {X 0,Y 392.762,Z 681.188,A -85,B 0,C 180,E1 11642.957,E2 11642.957} C_VEL
LIN {X 0,Y 401.014,Z 650.609,A -85,B 0,C 180,E1 11646.996,E2 11646.996} C_VEL
LIN {X 0,Y 409.18,Z 616.564,A -85,B 0,C 180,E1 11650.245,E2 11650.245} C_VEL
LIN {X 0,Y 416.139,Z 580.585,A -85,B 0,C 180,E1 11652.662,E2 11652.662} C_VEL
LIN {X 0,Y 420.6,Z 545.375,A -85,B 0,C 180,E1 11654.326,E2 11654.326} C_VEL
LIN {X 0,Y 402.251,Z 509.921,A -85,B 0,C 180,E1 11658.725,E2 11658.725} C_VEL
LIN {X 0,Y 383.887,Z 481.728,A -85,B 0,C 180,E1 11663.141,E2 11663.141} C_VEL
LIN {X 0,Y 374.413,Z 468.549,A -85,B 0,C 180,E1 11665.751,E2 11665.751} C_VEL
LIN {X 0,Y 371.613,Z 463.787,A -85,B 0,C 180,E1 11666.617,E2 11666.617} C_VEL
LIN {X 0,Y 371.518,Z 462.44,A -85,B 0,C 180,E1 11666.843,E2 11666.843} C_VEL
LIN {X 0,Y 371.717,Z 462.44,A -85,B 0,C 180,E1 11673.655,E2 11673.655} C_VEL
LIN {X 0,Y 372.027,Z 462.44,A -85,B 0,C 180,E1 11681.002,E2 11681.002} C_VEL
LIN {X 0,Y 372.353,Z 462.44,A -85,B 0,C 180,E1 11688.272,E2 11688.272} C_VEL
LIN {X 0,Y 372.739,Z 462.44,A -85,B 0,C 180,E1 11695.342,E2 11695.342} C_VEL
LIN {X 0,Y 372.919,Z 462.44,A -85,B 0,C 180,E1 11702.328,E2 11702.328} C_VEL
LIN {X 0,Y 372.406,Z 462.44,A -85,B 0,C 180,E1 11709.36,E2 11709.36} C_VEL
LIN {X 0,Y 372.103,Z 462.44,A -85,B 0,C 180,E1 11716.548,E2 11716.548} C_VEL
LIN {X 0,Y 371.87,Z 462.44,A -85,B 0,C 180,E1 11721.496,E2 11721.496} C_VEL
LIN {X 0,Y 371.65,Z 462.44,A -85,B 0,C 180,E1 11728.755,E2 11728.755} C_VEL
LIN {X 0,Y 373.705,Z 467.815,A -85,B 0,C 180,E1 11729.505,E2 11729.505} C_VEL
LIN {X 0,Y 376.57,Z 471.285,A -85,B 0,C 180,E1 11730.326,E2 11730.326} C_VEL
LIN {X 0,Y 392.938,Z 495.405,A -85,B 0,C 180,E1 11734.642,E2 11734.642} C_VEL
LIN {X 0,Y 410.051,Z 525.744,A -85,B 0,C 180,E1 11738.794,E2 11738.794} C_VEL
LIN {X 0,Y 420.869,Z 553.198,A -85,B 0,C 180,E1 11741.847,E2 11741.847} C_VEL
LIN {X 0,Y 414.847,Z 592.659,A -85,B 0,C 180,E1 11743.863,E2 11743.863} C_VEL
LIN {X 0,Y 407.448,Z 629.8,A -85,B 0,C 180,E1 11746.567,E2 11746.567} C_VEL
LIN {X 0,Y 399.014,Z 666.376,A -85,B 0,C 180,E1 11750.245,E2 11750.245} C_VEL
LIN {X 0,Y 390.715,Z 699.841,A -85,B 0,C 180,E1 11754.799,E2 11754.799} C_VEL
LIN {X 0,Y 383.911,Z 727.764,A -85,B 0,C 180,E1 11759.847,E2 11759.847} C_VEL
LIN {X 0,Y 378.498,Z 752.392,A -85,B 0,C 180,E1 11765.793,E2 11765.793} C_VEL
LIN {X 0,Y 375.311,Z 770.565,A -85,B 0,C 180,E1 11771.78,E2 11771.78} C_VEL
LIN {X 0,Y 373.526,Z 783.885,A -85,B 0,C 180,E1 11778.306,E2 11778.306} C_VEL
LIN {X 0,Y 373.147,Z 789.781,A -85,B 0,C 180,E1 11783.008,E2 11783.008} C_VEL
LIN {X 0,Y 373.013,Z 792.122,A -85,B 0,C 180,E1 11786.475,E2 11786.475} C_VEL
LIN {X 0,Y 370.497,Z 792.754,A -85,B 0,C 180,E1 11788.46,E2 11788.46} C_VEL
LIN {X 0,Y 365.087,Z 792.476,A -85,B 0,C 180,E1 11791.803,E2 11791.803} C_VEL
LIN {X 0,Y 365.261,Z 789.468,A -85,B 0,C 180,E1 11797.144,E2 11797.144} C_VEL
LIN {X 0,Y 366.003,Z 780.56,A -85,B 0,C 180,E1 11803.72,E2 11803.72} C_VEL
LIN {X 0,Y 368.01,Z 766.878,A -85,B 0,C 180,E1 11809.843,E2 11809.843} C_VEL
LIN {X 0,Y 371.892,Z 747.513,A -85,B 0,C 180,E1 11815.956,E2 11815.956} C_VEL
LIN {X 0,Y 377.815,Z 723.118,A -85,B 0,C 180,E1 11821.647,E2 11821.647} C_VEL
LIN {X 0,Y 385.566,Z 693.695,A -85,B 0,C 180,E1 11826.789,E2 11826.789} C_VEL
LIN {X 0,Y 393.911,Z 661.198,A -85,B 0,C 180,E1 11831.071,E2 11831.071} C_VEL
LIN {X 0,Y 402.972,Z 622.928,A -85,B 0,C 180,E1 11834.763,E2 11834.763} C_VEL
LIN {X 0,Y 410.903,Z 583.137,A -85,B 0,C 180,E1 11837.475,E2 11837.475} C_VEL
LIN {X 0,Y 414.532,Z 554.683,A -85,B 0,C 180,E1 11838.98,E2 11838.98} C_VEL
LIN {X 0,Y 403.922,Z 527.774,A -85,B 0,C 180,E1 11842.136,E2 11842.136} C_VEL
LIN {X 0,Y 387.53,Z 498.757,A -85,B 0,C 180,E1 11846.346,E2 11846.346} C_VEL
LIN {X 0,Y 371.695,Z 475.436,A -85,B 0,C 180,E1 11850.739,E2 11850.739} C_VEL
LIN {X 0,Y 367.222,Z 468.998,A -85,B 0,C 180,E1 11852.153,E2 11852.153} C_VEL
LIN {X 0,Y 363.964,Z 464.228,A -85,B 0,C 180,E1 11853.246,E2 11853.246} C_VEL
LIN {X 0,Y 363.809,Z 462.44,A -85,B 0,C 180,E1 11853.52,E2 11853.52} C_VEL
LIN {X 0,Y 364.061,Z 462.44,A -85,B 0,C 180,E1 11860.567,E2 11860.567} C_VEL
LIN {X 0,Y 364.236,Z 462.44,A -85,B 0,C 180,E1 11868.004,E2 11868.004} C_VEL
LIN {X 0,Y 364.753,Z 462.44,A -85,B 0,C 180,E1 11875.237,E2 11875.237} C_VEL
LIN {X 0,Y 365,Z 462.44,A -85,B 0,C 180,E1 11879.999,E2 11879.999} C_VEL
LIN {X 0,Y 364.602,Z 462.44,A -85,B 0,C 180,E1 11887.155,E2 11887.155} C_VEL
LIN {X 0,Y 364.217,Z 462.44,A -85,B 0,C 180,E1 11894.441,E2 11894.441} C_VEL
LIN {X 0,Y 363.847,Z 462.44,A -85,B 0,C 180,E1 11901.991,E2 11901.991} C_VEL
LIN {X 0,Y 363.639,Z 462.44,A -85,B 0,C 180,E1 11909.972,E2 11909.972} C_VEL
LIN {X 0,Y 363.66,Z 462.47,A -85,B 0,C 180,E1 11911.06,E2 11911.06} C_VEL
LIN {X 0,Y 365.571,Z 467.627,A -85,B 0,C 180,E1 11911.792,E2 11911.792} C_VEL
LIN {X 0,Y 368.784,Z 471.074,A -85,B 0,C 180,E1 11912.786,E2 11912.786} C_VEL
LIN {X 0,Y 386.243,Z 496.371,A -85,B 0,C 180,E1 11917.69,E2 11917.69} C_VEL
LIN {X 0,Y 404.147,Z 526.582,A -85,B 0,C 180,E1 11922.112,E2 11922.112} C_VEL
LIN {X 0,Y 415.093,Z 550.792,A -85,B 0,C 180,E1 11925.074,E2 11925.074} C_VEL
LIN {X 0,Y 409.259,Z 588.11,A -85,B 0,C 180,E1 11926.899,E2 11926.899} C_VEL
LIN {X 0,Y 401.538,Z 624.027,A -85,B 0,C 180,E1 11929.504,E2 11929.504} C_VEL
LIN {X 0,Y 392.957,Z 657.588,A -85,B 0,C 180,E1 11932.982,E2 11932.982} C_VEL
LIN {X 0,Y 384.473,Z 686.997,A -85,B 0,C 180,E1 11937.174,E2 11937.174} C_VEL
LIN {X 0,Y 376.828,Z 712.428,A -85,B 0,C 180,E1 11942.111,E2 11942.111} C_VEL
LIN {X 0,Y 371.381,Z 731.939,A -85,B 0,C 180,E1 11947.263,E2 11947.263} C_VEL
LIN {X 0,Y 367.682,Z 748.123,A -85,B 0,C 180,E1 11953.246,E2 11953.246} C_VEL
LIN {X 0,Y 365.904,Z 758.921,A -85,B 0,C 180,E1 11959.268,E2 11959.268} C_VEL
LIN {X 0,Y 365.194,Z 764.755,A -85,B 0,C 180,E1 11965.243,E2 11965.243} C_VEL
LIN {X 0,Y 365.24,Z 766.192,A -85,B 0,C 180,E1 11970,E2 11970} C_VEL
LIN {X 0,Y 365.254,Z 763.933,A -85,B 0,C 180,E1 11975.869,E2 11975.869} C_VEL
LIN {X 0,Y 366.178,Z 756.966,A -85,B 0,C 180,E1 11981.932,E2 11981.932} C_VEL
LIN {X 0,Y 368.294,Z 745.07,A -85,B 0,C 180,E1 11987.959,E2 11987.959} C_VEL
LIN {X 0,Y 372.641,Z 727.407,A -85,B 0,C 180,E1 11993.974,E2 11993.974} C_VEL
LIN {X 0,Y 378.958,Z 705.443,A -85,B 0,C 180,E1 11999.305,E2 11999.305} C_VEL
LIN {X 0,Y 386.889,Z 678.623,A -85,B 0,C 180,E1 12004.066,E2 12004.066} C_VEL
LIN {X 0,Y 395.274,Z 648.633,A -85,B 0,C 180,E1 12007.976,E2 12007.976} C_VEL
LIN {X 0,Y 403.785,Z 614.473,A -85,B 0,C 180,E1 12011.184,E2 12011.184} C_VEL
LIN {X 0,Y 410.807,Z 579.236,A -85,B 0,C 180,E1 12013.517,E2 12013.517} C_VEL
LIN {X 0,Y 414.811,Z 548.861,A -85,B 0,C 180,E1 12014.979,E2 12014.979} C_VEL
LIN {X 0,Y 398.172,Z 515.526,A -85,B 0,C 180,E1 12019.276,E2 12019.276} C_VEL
LIN {X 0,Y 380.318,Z 487.692,A -85,B 0,C 180,E1 12023.742,E2 12023.742} C_VEL
LIN {X 0,Y 370.459,Z 474.146,A -85,B 0,C 180,E1 12026.549,E2 12026.549} C_VEL
LIN {X 0,Y 366.88,Z 468.856,A -85,B 0,C 180,E1 12027.679,E2 12027.679} C_VEL
LIN {X 0,Y 363.759,Z 464.029,A -85,B 0,C 180,E1 12028.729,E2 12028.729} C_VEL
LIN {X 0,Y 363.633,Z 462.44,A -85,B 0,C 180,E1 12028.889,E2 12028.889} C_VEL
LIN {X 0,Y 363.83,Z 462.44,A -85,B 0,C 180,E1 12036.286,E2 12036.286} C_VEL
LIN {X 0,Y 364.246,Z 462.44,A -85,B 0,C 180,E1 12043.087,E2 12043.087} C_VEL
LIN {X 0,Y 364.511,Z 462.44,A -85,B 0,C 180,E1 12050.438,E2 12050.438} C_VEL
LIN {X 0,Y 364.951,Z 462.44,A -85,B 0,C 180,E1 12057.624,E2 12057.624} C_VEL
LIN {X 0,Y 365.002,Z 462.44,A -85,B 0,C 180,E1 12062.379,E2 12062.379} C_VEL
LIN {X 0,Y 364.466,Z 462.44,A -85,B 0,C 180,E1 12069.566,E2 12069.566} C_VEL
LIN {X 0,Y 364.133,Z 462.44,A -85,B 0,C 180,E1 12076.984,E2 12076.984} C_VEL
LIN {X 0,Y 363.798,Z 462.44,A -85,B 0,C 180,E1 12084.593,E2 12084.593} C_VEL
LIN {X 0,Y 363.785,Z 462.648,A -85,B 0,C 180,E1 12086.674,E2 12086.674} C_VEL
LIN {X 0,Y 365.845,Z 467.819,A -85,B 0,C 180,E1 12087.462,E2 12087.462} C_VEL
LIN {X 0,Y 368.888,Z 471.342,A -85,B 0,C 180,E1 12088.413,E2 12088.413} C_VEL
LIN {X 0,Y 385.608,Z 495.653,A -85,B 0,C 180,E1 12093.177,E2 12093.177} C_VEL
LIN {X 0,Y 402.794,Z 525.54,A -85,B 0,C 180,E1 12097.588,E2 12097.588} C_VEL
LIN {X 0,Y 413.555,Z 551.778,A -85,B 0,C 180,E1 12100.713,E2 12100.713} C_VEL
LIN {X 0,Y 414.863,Z 557.454,A -85,B 0,C 180,E1 12101.24,E2 12101.24} C_VEL
LIN {X 0,Y 407.817,Z 599.572,A -85,B 0,C 180,E1 12103.519,E2 12103.519} C_VEL
LIN {X 0,Y 399.438,Z 638.624,A -85,B 0,C 180,E1 12106.605,E2 12106.605} C_VEL
LIN {X 0,Y 390.178,Z 675.809,A -85,B 0,C 180,E1 12110.698,E2 12110.698} C_VEL
LIN {X 0,Y 381.693,Z 708.33,A -85,B 0,C 180,E1 12115.578,E2 12115.578} C_VEL
LIN {X 0,Y 374.423,Z 736.672,A -85,B 0,C 180,E1 12121.301,E2 12121.301} C_VEL
LIN {X 0,Y 369.61,Z 758.355,A -85,B 0,C 180,E1 12127.197,E2 12127.197} C_VEL
LIN {X 0,Y 366.807,Z 774.372,A -85,B 0,C 180,E1 12133.205,E2 12133.205} C_VEL
LIN {X 0,Y 365.532,Z 785.252,A -85,B 0,C 180,E1 12139.257,E2 12139.257} C_VEL
LIN {X 0,Y 365.168,Z 791.296,A -85,B 0,C 180,E1 12145.243,E2 12145.243} C_VEL
LIN {X 0,Y 365.241,Z 792.756,A -85,B 0,C 180,E1 12150,E2 12150} C_VEL
LIN {X 0,Y 365.087,Z 792.476,A -85,B 0,C 180,E1 12151.803,E2 12151.803} C_VEL
LIN {X 0,Y 362.559,Z 791.721,A -85,B 0,C 180,E1 12153.826,E2 12153.826} C_VEL
LIN {X 0,Y 357.386,Z 789.513,A -85,B 0,C 180,E1 12156.866,E2 12156.866} C_VEL
LIN {X 0,Y 357.348,Z 789.217,A -85,B 0,C 180,E1 12157.217,E2 12157.217} C_VEL
LIN {X 0,Y 358.069,Z 781.102,A -85,B 0,C 180,E1 12163.471,E2 12163.471} C_VEL
LIN {X 0,Y 360.017,Z 768.093,A -85,B 0,C 180,E1 12169.661,E2 12169.661} C_VEL
LIN {X 0,Y 363.877,Z 749.645,A -85,B 0,C 180,E1 12175.828,E2 12175.828} C_VEL
LIN {X 0,Y 370.197,Z 725.021,A -85,B 0,C 180,E1 12181.845,E2 12181.845} C_VEL
LIN {X 0,Y 378.441,Z 695.211,A -85,B 0,C 180,E1 12187.24,E2 12187.24} C_VEL
LIN {X 0,Y 387.649,Z 660.925,A -85,B 0,C 180,E1 12191.845,E2 12191.845} C_VEL
LIN {X 0,Y 396.932,Z 623.506,A -85,B 0,C 180,E1 12195.498,E2 12195.498} C_VEL
LIN {X 0,Y 405.203,Z 583.794,A -85,B 0,C 180,E1 12198.237,E2 12198.237} C_VEL
LIN {X 0,Y 408.84,Z 557.969,A -85,B 0,C 180,E1 12199.628,E2 12199.628} C_VEL
LIN {X 0,Y 398.771,Z 531.935,A -85,B 0,C 180,E1 12202.801,E2 12202.801} C_VEL
LIN {X 0,Y 383.335,Z 503.976,A -85,B 0,C 180,E1 12207.023,E2 12207.023} C_VEL
LIN {X 0,Y 368.476,Z 481.825,A -85,B 0,C 180,E1 12211.318,E2 12211.318} C_VEL
LIN {X 0,Y 363.001,Z 474.445,A -85,B 0,C 180,E1 12213.095,E2 12213.095} C_VEL
LIN {X 0,Y 359.363,Z 468.962,A -85,B 0,C 180,E1 12214.392,E2 12214.392} C_VEL
LIN {X 0,Y 356.115,Z 464.21,A -85,B 0,C 180,E1 12215.614,E2 12215.614} C_VEL
LIN {X 0,Y 355.929,Z 462.44,A -85,B 0,C 180,E1 12215.934,E2 12215.934} C_VEL
LIN {X 0,Y 356.182,Z 462.44,A -85,B 0,C 180,E1 12222.689,E2 12222.689} C_VEL
LIN {X 0,Y 356.464,Z 462.44,A -85,B 0,C 180,E1 12230.217,E2 12230.217} C_VEL
LIN {X 0,Y 357.112,Z 462.44,A -85,B 0,C 180,E1 12237.569,E2 12237.569} C_VEL
LIN {X 0,Y 356.842,Z 462.44,A -85,B 0,C 180,E1 12244.866,E2 12244.866} C_VEL
LIN {X 0,Y 356.418,Z 462.44,A -85,B 0,C 180,E1 12252.289,E2 12252.289} C_VEL
LIN {X 0,Y 356.04,Z 462.44,A -85,B 0,C 180,E1 12259.886,E2 12259.886} C_VEL
LIN {X 0,Y 355.746,Z 462.44,A -85,B 0,C 180,E1 12267.911,E2 12267.911} C_VEL
LIN {X 0,Y 355.811,Z 463.279,A -85,B 0,C 180,E1 12268.703,E2 12268.703} C_VEL
LIN {X 0,Y 358.423,Z 468.375,A -85,B 0,C 180,E1 12269.737,E2 12269.737} C_VEL
LIN {X 0,Y 360.939,Z 470.864,A -85,B 0,C 180,E1 12270.595,E2 12270.595} C_VEL
LIN {X 0,Y 376.393,Z 493.058,A -85,B 0,C 180,E1 12275.418,E2 12275.418} C_VEL
LIN {X 0,Y 392.332,Z 518.208,A -85,B 0,C 180,E1 12279.624,E2 12279.624} C_VEL
LIN {X 0,Y 408.123,Z 550.029,A -85,B 0,C 180,E1 12283.96,E2 12283.96} C_VEL
LIN {X 0,Y 409.3,Z 554.017,A -85,B 0,C 180,E1 12284.381,E2 12284.381} C_VEL
LIN {X 0,Y 403.124,Z 590.958,A -85,B 0,C 180,E1 12286.264,E2 12286.264} C_VEL
LIN {X 0,Y 395.042,Z 626.476,A -85,B 0,C 180,E1 12288.923,E2 12288.923} C_VEL
LIN {X 0,Y 386.296,Z 659.171,A -85,B 0,C 180,E1 12292.411,E2 12292.411} C_VEL
LIN {X 0,Y 377.777,Z 687.361,A -85,B 0,C 180,E1 12296.508,E2 12296.508} C_VEL
LIN {X 0,Y 369.722,Z 712.795,A -85,B 0,C 180,E1 12301.526,E2 12301.526} C_VEL
LIN {X 0,Y 363.794,Z 732.812,A -85,B 0,C 180,E1 12306.946,E2 12306.946} C_VEL
LIN {X 0,Y 359.994,Z 748.445,A -85,B 0,C 180,E1 12312.877,E2 12312.877} C_VEL
LIN {X 0,Y 358.083,Z 759.225,A -85,B 0,C 180,E1 12319.031,E2 12319.031} C_VEL
LIN {X 0,Y 357.301,Z 765.047,A -85,B 0,C 180,E1 12325.138,E2 12325.138} C_VEL
LIN {X 0,Y 357.343,Z 766.479,A -85,B 0,C 180,E1 12330,E2 12330} C_VEL
LIN {X 0,Y 357.318,Z 764.984,A -85,B 0,C 180,E1 12334.862,E2 12334.862} C_VEL
LIN {X 0,Y 358.101,Z 759.103,A -85,B 0,C 180,E1 12340.969,E2 12340.969} C_VEL
LIN {X 0,Y 360.321,Z 746.866,A -85,B 0,C 180,E1 12347.738,E2 12347.738} C_VEL
LIN {X 0,Y 364.433,Z 730.827,A -85,B 0,C 180,E1 12353.591,E2 12353.591} C_VEL
LIN {X 0,Y 371.077,Z 708.647,A -85,B 0,C 180,E1 12359.317,E2 12359.317} C_VEL
LIN {X 0,Y 379.669,Z 681.039,A -85,B 0,C 180,E1 12364.436,E2 12364.436} C_VEL
LIN {X 0,Y 388.68,Z 650.383,A -85,B 0,C 180,E1 12368.557,E2 12368.557} C_VEL
LIN {X 0,Y 397.518,Z 616.611,A -85,B 0,C 180,E1 12371.813,E2 12371.813} C_VEL
LIN {X 0,Y 404.973,Z 581.07,A -85,B 0,C 180,E1 12374.229,E2 12374.229} C_VEL
LIN {X 0,Y 408.947,Z 552.115,A -85,B 0,C 180,E1 12375.685,E2 12375.685} C_VEL
LIN {X 0,Y 393.505,Z 520.267,A -85,B 0,C 180,E1 12379.953,E2 12379.953} C_VEL
LIN {X 0,Y 377.09,Z 493.998,A -85,B 0,C 180,E1 12384.273,E2 12384.273} C_VEL
LIN {X 0,Y 363.744,Z 475.319,A -85,B 0,C 180,E1 12388.304,E2 12388.304} C_VEL
LIN {X 0,Y 359.506,Z 469.197,A -85,B 0,C 180,E1 12389.768,E2 12389.768} C_VEL
LIN {X 0,Y 355.941,Z 464.191,A -85,B 0,C 180,E1 12391.084,E2 12391.084} C_VEL
LIN {X 0,Y 355.717,Z 462.44,A -85,B 0,C 180,E1 12391.406,E2 12391.406} C_VEL
LIN {X 0,Y 356.01,Z 462.44,A -85,B 0,C 180,E1 12399.338,E2 12399.338} C_VEL
LIN {X 0,Y 356.371,Z 462.44,A -85,B 0,C 180,E1 12405.234,E2 12405.234} C_VEL
LIN {X 0,Y 356.731,Z 462.44,A -85,B 0,C 180,E1 12412.687,E2 12412.687} C_VEL
LIN {X 0,Y 357.176,Z 462.44,A -85,B 0,C 180,E1 12420.001,E2 12420.001} C_VEL
LIN {X 0,Y 356.754,Z 462.44,A -85,B 0,C 180,E1 12427.316,E2 12427.316} C_VEL
LIN {X 0,Y 356.273,Z 462.44,A -85,B 0,C 180,E1 12434.773,E2 12434.773} C_VEL
LIN {X 0,Y 355.949,Z 462.44,A -85,B 0,C 180,E1 12442.508,E2 12442.508} C_VEL
LIN {X 0,Y 355.923,Z 462.452,A -85,B 0,C 180,E1 12444.29,E2 12444.29} C_VEL
LIN {X 0,Y 357.617,Z 467.385,A -85,B 0,C 180,E1 12445.047,E2 12445.047} C_VEL
LIN {X 0,Y 361.09,Z 471.144,A -85,B 0,C 180,E1 12446.253,E2 12446.253} C_VEL
LIN {X 0,Y 375.52,Z 492.046,A -85,B 0,C 180,E1 12450.826,E2 12450.826} C_VEL
LIN {X 0,Y 391.356,Z 517.557,A -85,B 0,C 180,E1 12455.162,E2 12455.162} C_VEL
LIN {X 0,Y 404.95,Z 546.384,A -85,B 0,C 180,E1 12459.057,E2 12459.057} C_VEL
LIN {X 0,Y 408.949,Z 560.224,A -85,B 0,C 180,E1 12460.557,E2 12460.557} C_VEL
LIN {X 0,Y 401.888,Z 600.578,A -85,B 0,C 180,E1 12462.797,E2 12462.797} C_VEL
LIN {X 0,Y 393.385,Z 638.679,A -85,B 0,C 180,E1 12465.848,E2 12465.848} C_VEL
LIN {X 0,Y 383.906,Z 674.982,A -85,B 0,C 180,E1 12469.869,E2 12469.869} C_VEL
LIN {X 0,Y 374.707,Z 708.358,A -85,B 0,C 180,E1 12474.942,E2 12474.942} C_VEL
LIN {X 0,Y 367.206,Z 736.264,A -85,B 0,C 180,E1 12480.682,E2 12480.682} C_VEL
LIN {X 0,Y 361.848,Z 758.853,A -85,B 0,C 180,E1 12486.998,E2 12486.998} C_VEL
LIN {X 0,Y 358.84,Z 775.351,A -85,B 0,C 180,E1 12493.452,E2 12493.452} C_VEL
LIN {X 0,Y 357.646,Z 784.906,A -85,B 0,C 180,E1 12499.017,E2 12499.017} C_VEL
LIN {X 0,Y 357.271,Z 790.996,A -85,B 0,C 180,E1 12505.138,E2 12505.138} C_VEL
LIN {X 0,Y 357.344,Z 792.469,A -85,B 0,C 180,E1 12510,E2 12510} C_VEL
LIN {X 0,Y 357.252,Z 790.996,A -85,B 0,C 180,E1 12514.862,E2 12514.862} C_VEL
LIN {X 0,Y 357.348,Z 789.217,A -85,B 0,C 180,E1 12517.217,E2 12517.217} C_VEL
LIN {X 0,Y 355.077,Z 787.255,A -85,B 0,C 180,E1 12519.269,E2 12519.269} C_VEL
LIN {X 0,Y 350.063,Z 783.083,A -85,B 0,C 180,E1 12522.33,E2 12522.33} C_VEL
LIN {X 0,Y 350.026,Z 782.523,A -85,B 0,C 180,E1 12522.68,E2 12522.68} C_VEL
LIN {X 0,Y 351.996,Z 769.66,A -85,B 0,C 180,E1 12529.342,E2 12529.342} C_VEL
LIN {X 0,Y 356.253,Z 750.195,A -85,B 0,C 180,E1 12536.143,E2 12536.143} C_VEL
LIN {X 0,Y 363.14,Z 724.499,A -85,B 0,C 180,E1 12542.564,E2 12542.564} C_VEL
LIN {X 0,Y 371.857,Z 694.797,A -85,B 0,C 180,E1 12548.008,E2 12548.008} C_VEL
LIN {X 0,Y 381.573,Z 660.413,A -85,B 0,C 180,E1 12552.667,E2 12552.667} C_VEL
LIN {X 0,Y 391.277,Z 622.552,A -85,B 0,C 180,E1 12556.384,E2 12556.384} C_VEL
LIN {X 0,Y 399.863,Z 582.816,A -85,B 0,C 180,E1 12559.113,E2 12559.113} C_VEL
LIN {X 0,Y 403.054,Z 560.908,A -85,B 0,C 180,E1 12560.314,E2 12560.314} C_VEL
LIN {X 0,Y 393.031,Z 534.844,A -85,B 0,C 180,E1 12563.664,E2 12563.664} C_VEL
LIN {X 0,Y 377.861,Z 506.776,A -85,B 0,C 180,E1 12568.103,E2 12568.103} C_VEL
LIN {X 0,Y 361.62,Z 482.672,A -85,B 0,C 180,E1 12573.146,E2 12573.146} C_VEL
LIN {X 0,Y 355.799,Z 475.054,A -85,B 0,C 180,E1 12575.223,E2 12575.223} C_VEL
LIN {X 0,Y 352.063,Z 469.321,A -85,B 0,C 180,E1 12576.713,E2 12576.713} C_VEL
LIN {X 0,Y 348.331,Z 464.509,A -85,B 0,C 180,E1 12578.279,E2 12578.279} C_VEL
LIN {X 0,Y 348.034,Z 462.44,A -85,B 0,C 180,E1 12578.614,E2 12578.614} C_VEL
LIN {X 0,Y 348.247,Z 462.44,A -85,B 0,C 180,E1 12584.879,E2 12584.879} C_VEL
LIN {X 0,Y 348.8,Z 462.44,A -85,B 0,C 180,E1 12592.517,E2 12592.517} C_VEL
LIN {X 0,Y 349.211,Z 462.44,A -85,B 0,C 180,E1 12599.999,E2 12599.999} C_VEL
LIN {X 0,Y 348.748,Z 462.44,A -85,B 0,C 180,E1 12607.482,E2 12607.482} C_VEL
LIN {X 0,Y 348.313,Z 462.44,A -85,B 0,C 180,E1 12615.116,E2 12615.116} C_VEL
LIN {X 0,Y 347.907,Z 462.44,A -85,B 0,C 180,E1 12623.055,E2 12623.055} C_VEL
LIN {X 0,Y 347.834,Z 462.62,A -85,B 0,C 180,E1 12625.893,E2 12625.893} C_VEL
LIN {X 0,Y 349.794,Z 467.662,A -85,B 0,C 180,E1 12626.849,E2 12626.849} C_VEL
LIN {X 0,Y 353.288,Z 471.024,A -85,B 0,C 180,E1 12628.21,E2 12628.21} C_VEL
LIN {X 0,Y 368.072,Z 491.677,A -85,B 0,C 180,E1 12633.333,E2 12633.333} C_VEL
LIN {X 0,Y 385.288,Z 518.446,A -85,B 0,C 180,E1 12638.243,E2 12638.243} C_VEL
LIN {X 0,Y 400.593,Z 549.096,A -85,B 0,C 180,E1 12642.679,E2 12642.679} C_VEL
LIN {X 0,Y 403.624,Z 556.263,A -85,B 0,C 180,E1 12643.619,E2 12643.619} C_VEL
LIN {X 0,Y 396.684,Z 595.773,A -85,B 0,C 180,E1 12645.739,E2 12645.739} C_VEL
LIN {X 0,Y 387.905,Z 631.956,A -85,B 0,C 180,E1 12648.614,E2 12648.614} C_VEL
LIN {X 0,Y 377.936,Z 666.192,A -85,B 0,C 180,E1 12652.522,E2 12652.522} C_VEL
LIN {X 0,Y 368.509,Z 695.575,A -85,B 0,C 180,E1 12657.221,E2 12657.221} C_VEL
LIN {X 0,Y 360.599,Z 719.532,A -85,B 0,C 180,E1 12662.491,E2 12662.491} C_VEL
LIN {X 0,Y 354.663,Z 739.674,A -85,B 0,C 180,E1 12668.723,E2 12668.723} C_VEL
LIN {X 0,Y 351.272,Z 753.649,A -85,B 0,C 180,E1 12675.011,E2 12675.011} C_VEL
LIN {X 0,Y 349.841,Z 762.396,A -85,B 0,C 180,E1 12681.287,E2 12681.287} C_VEL
LIN {X 0,Y 349.341,Z 766.415,A -85,B 0,C 180,E1 12687.516,E2 12687.516} C_VEL
LIN {X 0,Y 349.42,Z 766.376,A -85,B 0,C 180,E1 12692.484,E2 12692.484} C_VEL
LIN {X 0,Y 349.853,Z 762.311,A -85,B 0,C 180,E1 12698.713,E2 12698.713} C_VEL
LIN {X 0,Y 351.501,Z 752.39,A -85,B 0,C 180,E1 12705.618,E2 12705.618} C_VEL
LIN {X 0,Y 355.136,Z 737.779,A -85,B 0,C 180,E1 12711.904,E2 12711.904} C_VEL
LIN {X 0,Y 361.401,Z 717.023,A -85,B 0,C 180,E1 12718.062,E2 12718.062} C_VEL
LIN {X 0,Y 370.022,Z 690.933,A -85,B 0,C 180,E1 12723.533,E2 12723.533} C_VEL
LIN {X 0,Y 379.471,Z 661.255,A -85,B 0,C 180,E1 12728.023,E2 12728.023} C_VEL
LIN {X 0,Y 388.482,Z 629.657,A -85,B 0,C 180,E1 12731.497,E2 12731.497} C_VEL
LIN {X 0,Y 396.76,Z 594.545,A -85,B 0,C 180,E1 12734.263,E2 12734.263} C_VEL
LIN {X 0,Y 403.337,Z 555.69,A -85,B 0,C 180,E1 12736.359,E2 12736.359} C_VEL
LIN {X 0,Y 388.178,Z 523.571,A -85,B 0,C 180,E1 12740.828,E2 12740.828} C_VEL
LIN {X 0,Y 370.737,Z 495.495,A -85,B 0,C 180,E1 12745.74,E2 12745.74} C_VEL
LIN {X 0,Y 356.729,Z 476.022,A -85,B 0,C 180,E1 12750.338,E2 12750.338} C_VEL
LIN {X 0,Y 351.8,Z 469.291,A -85,B 0,C 180,E1 12752.232,E2 12752.232} C_VEL
LIN {X 0,Y 348.129,Z 464.577,A -85,B 0,C 180,E1 12753.758,E2 12753.758} C_VEL
LIN {X 0,Y 347.867,Z 462.44,A -85,B 0,C 180,E1 12754.017,E2 12754.017} C_VEL
LIN {X 0,Y 348.326,Z 462.44,A -85,B 0,C 180,E1 12762.289,E2 12762.289} C_VEL
LIN {X 0,Y 348.64,Z 462.44,A -85,B 0,C 180,E1 12769.999,E2 12769.999} C_VEL
LIN {X 0,Y 349.156,Z 462.44,A -85,B 0,C 180,E1 12777.516,E2 12777.516} C_VEL
LIN {X 0,Y 349.02,Z 462.44,A -85,B 0,C 180,E1 12783.802,E2 12783.802} C_VEL
LIN {X 0,Y 348.591,Z 462.44,A -85,B 0,C 180,E1 12790.006,E2 12790.006} C_VEL
LIN {X 0,Y 348.247,Z 462.44,A -85,B 0,C 180,E1 12797.718,E2 12797.718} C_VEL
LIN {X 0,Y 348.084,Z 463.142,A -85,B 0,C 180,E1 12801.617,E2 12801.617} C_VEL
LIN {X 0,Y 350.549,Z 468.18,A -85,B 0,C 180,E1 12802.756,E2 12802.756} C_VEL
LIN {X 0,Y 353.371,Z 470.999,A -85,B 0,C 180,E1 12803.852,E2 12803.852} C_VEL
LIN {X 0,Y 367.758,Z 491.6,A -85,B 0,C 180,E1 12808.906,E2 12808.906} C_VEL
LIN {X 0,Y 384.122,Z 517.389,A -85,B 0,C 180,E1 12813.72,E2 12813.72} C_VEL
LIN {X 0,Y 398.241,Z 546.887,A -85,B 0,C 180,E1 12817.981,E2 12817.981} C_VEL
LIN {X 0,Y 403.066,Z 563.368,A -85,B 0,C 180,E1 12819.876,E2 12819.876} C_VEL
LIN {X 0,Y 395.776,Z 602.673,A -85,B 0,C 180,E1 12822.128,E2 12822.128} C_VEL
LIN {X 0,Y 386.943,Z 640.349,A -85,B 0,C 180,E1 12825.223,E2 12825.223} C_VEL
LIN {X 0,Y 377.147,Z 676.106,A -85,B 0,C 180,E1 12829.278,E2 12829.278} C_VEL
LIN {X 0,Y 367.874,Z 708.201,A -85,B 0,C 180,E1 12834.25,E2 12834.25} C_VEL
LIN {X 0,Y 360.018,Z 735.874,A -85,B 0,C 180,E1 12840.038,E2 12840.038} C_VEL
LIN {X 0,Y 354.296,Z 758.485,A -85,B 0,C 180,E1 12846.478,E2 12846.478} C_VEL
LIN {X 0,Y 351.059,Z 775,A -85,B 0,C 180,E1 12853.074,E2 12853.074} C_VEL
LIN {X 0,Y 349.772,Z 784.57,A -85,B 0,C 180,E1 12858.767,E2 12858.767} C_VEL
LIN {X 0,Y 349.373,Z 790.696,A -85,B 0,C 180,E1 12865.027,E2 12865.027} C_VEL
LIN {X 0,Y 349.446,Z 792.182,A -85,B 0,C 180,E1 12870,E2 12870} C_VEL
LIN {X 0,Y 349.367,Z 790.697,A -85,B 0,C 180,E1 12874.973,E2 12874.973} C_VEL
LIN {X 0,Y 349.788,Z 784.571,A -85,B 0,C 180,E1 12881.233,E2 12881.233} C_VEL
LIN {X 0,Y 350.026,Z 782.523,A -85,B 0,C 180,E1 12882.68,E2 12882.68} C_VEL
LIN {X 0,Y 349.034,Z 780.339,A -85,B 0,C 180,E1 12884.059,E2 12884.059} C_VEL
LIN {X 0,Y 343.578,Z 773.604,A -85,B 0,C 180,E1 12887.818,E2 12887.818} C_VEL
LIN {X 0,Y 343.629,Z 772.854,A -85,B 0,C 180,E1 12888.164,E2 12888.164} C_VEL
LIN {X 0,Y 347.17,Z 756.208,A -85,B 0,C 180,E1 12894.718,E2 12894.718} C_VEL
LIN {X 0,Y 353.517,Z 733.13,A -85,B 0,C 180,E1 12901.218,E2 12901.218} C_VEL
LIN {X 0,Y 362.135,Z 704.546,A -85,B 0,C 180,E1 12907.107,E2 12907.107} C_VEL
LIN {X 0,Y 372.039,Z 672.293,A -85,B 0,C 180,E1 12911.988,E2 12911.988} C_VEL
LIN {X 0,Y 382.247,Z 635.843,A -85,B 0,C 180,E1 12916.028,E2 12916.028} C_VEL
LIN {X 0,Y 391.635,Z 596.456,A -85,B 0,C 180,E1 12919.131,E2 12919.131} C_VEL
LIN {X 0,Y 397.384,Z 564.272,A -85,B 0,C 180,E1 12920.981,E2 12920.981} C_VEL
LIN {X 0,Y 387.818,Z 538.714,A -85,B 0,C 180,E1 12924.412,E2 12924.412} C_VEL
LIN {X 0,Y 373.894,Z 512.231,A -85,B 0,C 180,E1 12928.781,E2 12928.781} C_VEL
LIN {X 0,Y 358.664,Z 489.186,A -85,B 0,C 180,E1 12933.729,E2 12933.729} C_VEL
LIN {X 0,Y 349.221,Z 476.132,A -85,B 0,C 180,E1 12937.37,E2 12937.37} C_VEL
LIN {X 0,Y 345.481,Z 470.209,A -85,B 0,C 180,E1 12939.057,E2 12939.057} C_VEL
LIN {X 0,Y 340.739,Z 465.291,A -85,B 0,C 180,E1 12941.291,E2 12941.291} C_VEL
LIN {X 0,Y 340.262,Z 462.44,A -85,B 0,C 180,E1 12941.852,E2 12941.852} C_VEL
LIN {X 0,Y 340.579,Z 462.44,A -85,B 0,C 180,E1 12949.756,E2 12949.756} C_VEL
LIN {X 0,Y 341.288,Z 462.44,A -85,B 0,C 180,E1 12957.456,E2 12957.456} C_VEL
LIN {X 0,Y 341.182,Z 462.44,A -85,B 0,C 180,E1 12962.542,E2 12962.542} C_VEL
LIN {X 0,Y 340.652,Z 462.44,A -85,B 0,C 180,E1 12970.239,E2 12970.239} C_VEL
LIN {X 0,Y 340.26,Z 462.44,A -85,B 0,C 180,E1 12978.146,E2 12978.146} C_VEL
LIN {X 0,Y 339.997,Z 462.651,A -85,B 0,C 180,E1 12982.67,E2 12982.67} C_VEL
LIN {X 0,Y 341.961,Z 467.698,A -85,B 0,C 180,E1 12983.807,E2 12983.807} C_VEL
LIN {X 0,Y 345.572,Z 471.018,A -85,B 0,C 180,E1 12985.445,E2 12985.445} C_VEL
LIN {X 0,Y 350.032,Z 476.822,A -85,B 0,C 180,E1 12987.357,E2 12987.357} C_VEL
LIN {X 0,Y 365.274,Z 498.411,A -85,B 0,C 180,E1 12992.841,E2 12992.841} C_VEL
LIN {X 0,Y 381.455,Z 524.476,A -85,B 0,C 180,E1 12997.737,E2 12997.737} C_VEL
LIN {X 0,Y 396.471,Z 555.886,A -85,B 0,C 180,E1 13002.408,E2 13002.408} C_VEL
LIN {X 0,Y 397.836,Z 560.497,A -85,B 0,C 180,E1 13002.961,E2 13002.961} C_VEL
LIN {X 0,Y 390.752,Z 597.779,A -85,B 0,C 180,E1 13005.025,E2 13005.025} C_VEL
LIN {X 0,Y 381.924,Z 632.596,A -85,B 0,C 180,E1 13007.837,E2 13007.837} C_VEL
LIN {X 0,Y 371.609,Z 666.613,A -85,B 0,C 180,E1 13011.77,E2 13011.77} C_VEL
LIN {X 0,Y 362.093,Z 695.038,A -85,B 0,C 180,E1 13016.354,E2 13016.354} C_VEL
LIN {X 0,Y 353.427,Z 719.878,A -85,B 0,C 180,E1 13021.884,E2 13021.884} C_VEL
LIN {X 0,Y 347.121,Z 740,A -85,B 0,C 180,E1 13028.237,E2 13028.237} C_VEL
LIN {X 0,Y 343.535,Z 753.956,A -85,B 0,C 180,E1 13034.666,E2 13034.666} C_VEL
LIN {X 0,Y 341.997,Z 762.689,A -85,B 0,C 180,E1 13041.086,E2 13041.086} C_VEL
LIN {X 0,Y 341.458,Z 766.703,A -85,B 0,C 180,E1 13047.459,E2 13047.459} C_VEL
LIN {X 0,Y 341.531,Z 766.664,A -85,B 0,C 180,E1 13052.541,E2 13052.541} C_VEL
LIN {X 0,Y 342.011,Z 762.605,A -85,B 0,C 180,E1 13058.914,E2 13058.914} C_VEL
LIN {X 0,Y 343.781,Z 752.703,A -85,B 0,C 180,E1 13065.978,E2 13065.978} C_VEL
LIN {X 0,Y 347.645,Z 738.108,A -85,B 0,C 180,E1 13072.402,E2 13072.402} C_VEL
LIN {X 0,Y 354.31,Z 717.384,A -85,B 0,C 180,E1 13078.675,E2 13078.675} C_VEL
LIN {X 0,Y 363.36,Z 691.329,A -85,B 0,C 180,E1 13084.232,E2 13084.232} C_VEL
LIN {X 0,Y 373.192,Z 661.71,A -85,B 0,C 180,E1 13088.781,E2 13088.781} C_VEL
LIN {X 0,Y 382.951,Z 628.705,A -85,B 0,C 180,E1 13092.425,E2 13092.425} C_VEL
LIN {X 0,Y 391.796,Z 592.35,A -85,B 0,C 180,E1 13095.245,E2 13095.245} C_VEL
LIN {X 0,Y 397.539,Z 559.036,A -85,B 0,C 180,E1 13097.092,E2 13097.092} C_VEL
LIN {X 0,Y 383.765,Z 528.601,A -85,B 0,C 180,E1 13101.476,E2 13101.476} C_VEL
LIN {X 0,Y 367.111,Z 501.213,A -85,B 0,C 180,E1 13106.456,E2 13106.456} C_VEL
LIN {X 0,Y 353.78,Z 482.517,A -85,B 0,C 180,E1 13111,E2 13111} C_VEL
LIN {X 0,Y 349.169,Z 476.183,A -85,B 0,C 180,E1 13112.832,E2 13112.832} C_VEL
LIN {X 0,Y 345.346,Z 470.27,A -85,B 0,C 180,E1 13114.534,E2 13114.534} C_VEL
LIN {X 0,Y 340.569,Z 465.288,A -85,B 0,C 180,E1 13116.765,E2 13116.765} C_VEL
LIN {X 0,Y 340.05,Z 462.44,A -85,B 0,C 180,E1 13117.247,E2 13117.247} C_VEL
LIN {X 0,Y 340.512,Z 462.44,A -85,B 0,C 180,E1 13124.53,E2 13124.53} C_VEL
LIN {X 0,Y 340.866,Z 462.44,A -85,B 0,C 180,E1 13132.344,E2 13132.344} C_VEL
LIN {X 0,Y 341.385,Z 462.44,A -85,B 0,C 180,E1 13140.001,E2 13140.001} C_VEL
LIN {X 0,Y 340.876,Z 462.44,A -85,B 0,C 180,E1 13147.658,E2 13147.658} C_VEL
LIN {X 0,Y 340.392,Z 462.44,A -85,B 0,C 180,E1 13155.479,E2 13155.479} C_VEL
LIN {X 0,Y 340.256,Z 462.467,A -85,B 0,C 180,E1 13158.401,E2 13158.401} C_VEL
LIN {X 0,Y 341.9,Z 467.321,A -85,B 0,C 180,E1 13159.398,E2 13159.398} C_VEL
LIN {X 0,Y 345.793,Z 471.243,A -85,B 0,C 180,E1 13161.175,E2 13161.175} C_VEL
LIN {X 0,Y 351.769,Z 479.808,A -85,B 0,C 180,E1 13163.734,E2 13163.734} C_VEL
LIN {X 0,Y 360.676,Z 492.072,A -85,B 0,C 180,E1 13167.013,E2 13167.013} C_VEL
LIN {X 0,Y 376.101,Z 516.007,A -85,B 0,C 180,E1 13171.926,E2 13171.926} C_VEL
LIN {X 0,Y 390.17,Z 544.084,A -85,B 0,C 180,E1 13176.368,E2 13176.368} C_VEL
LIN {X 0,Y 397.462,Z 564.774,A -85,B 0,C 180,E1 13179.082,E2 13179.082} C_VEL
LIN {X 0,Y 389.948,Z 603.87,A -85,B 0,C 180,E1 13181.376,E2 13181.376} C_VEL
LIN {X 0,Y 381.167,Z 639.812,A -85,B 0,C 180,E1 13184.355,E2 13184.355} C_VEL
LIN {X 0,Y 370.931,Z 675.647,A -85,B 0,C 180,E1 13188.446,E2 13188.446} C_VEL
LIN {X 0,Y 360.993,Z 708.305,A -85,B 0,C 180,E1 13193.576,E2 13193.576} C_VEL
LIN {X 0,Y 352.829,Z 735.492,A -85,B 0,C 180,E1 13199.362,E2 13199.362} C_VEL
LIN {X 0,Y 347.091,Z 756.926,A -85,B 0,C 180,E1 13205.518,E2 13205.518} C_VEL
LIN {X 0,Y 343.3,Z 774.664,A -85,B 0,C 180,E1 13212.68,E2 13212.68} C_VEL
LIN {X 0,Y 341.921,Z 784.256,A -85,B 0,C 180,E1 13218.505,E2 13218.505} C_VEL
LIN {X 0,Y 341.466,Z 790.4,A -85,B 0,C 180,E1 13224.912,E2 13224.912} C_VEL
LIN {X 0,Y 341.575,Z 791.895,A -85,B 0,C 180,E1 13230,E2 13230} C_VEL
LIN {X 0,Y 341.46,Z 790.4,A -85,B 0,C 180,E1 13235.088,E2 13235.088} C_VEL
LIN {X 0,Y 341.934,Z 784.257,A -85,B 0,C 180,E1 13241.494,E2 13241.494} C_VEL
LIN {X 0,Y 343.629,Z 772.854,A -85,B 0,C 180,E1 13248.164,E2 13248.164} C_VEL
LIN {X 0,Y 342.965,Z 769.992,A -85,B 0,C 180,E1 13249.537,E2 13249.537} C_VEL
LIN {X 0,Y 338.386,Z 761.456,A -85,B 0,C 180,E1 13253.286,E2 13253.286} C_VEL
LIN {X 0,Y 338.533,Z 760.54,A -85,B 0,C 180,E1 13253.625,E2 13253.625} C_VEL
LIN {X 0,Y 344.426,Z 739.177,A -85,B 0,C 180,E1 13260.283,E2 13260.283} C_VEL
LIN {X 0,Y 352.848,Z 712.79,A -85,B 0,C 180,E1 13266.279,E2 13266.279} C_VEL
LIN {X 0,Y 362.536,Z 682.707,A -85,B 0,C 180,E1 13271.351,E2 13271.351} C_VEL
LIN {X 0,Y 373.049,Z 647.896,A -85,B 0,C 180,E1 13275.673,E2 13275.673} C_VEL
LIN {X 0,Y 383.056,Z 610.125,A -85,B 0,C 180,E1 13279.041,E2 13279.041} C_VEL
LIN {X 0,Y 391.531,Z 569.43,A -85,B 0,C 180,E1 13281.57,E2 13281.57} C_VEL
LIN {X 0,Y 387.526,Z 554.313,A -85,B 0,C 180,E1 13283.431,E2 13283.431} C_VEL
LIN {X 0,Y 374.247,Z 525.369,A -85,B 0,C 180,E1 13288.014,E2 13288.014} C_VEL
LIN {X 0,Y 359.881,Z 501.686,A -85,B 0,C 180,E1 13292.843,E2 13292.843} C_VEL
LIN {X 0,Y 347.358,Z 483.592,A -85,B 0,C 180,E1 13297.665,E2 13297.665} C_VEL
LIN {X 0,Y 341.785,Z 476.385,A -85,B 0,C 180,E1 13300.201,E2 13300.201} C_VEL
LIN {X 0,Y 338.12,Z 470.799,A -85,B 0,C 180,E1 13302.134,E2 13302.134} C_VEL
LIN {X 0,Y 332.778,Z 464.916,A -85,B 0,C 180,E1 13305.256,E2 13305.256} C_VEL
LIN {X 0,Y 332.398,Z 462.44,A -85,B 0,C 180,E1 13305.828,E2 13305.828} C_VEL
LIN {X 0,Y 332.92,Z 462.44,A -85,B 0,C 180,E1 13312.158,E2 13312.158} C_VEL
LIN {X 0,Y 333.387,Z 462.44,A -85,B 0,C 180,E1 13317.663,E2 13317.663} C_VEL
LIN {X 0,Y 333.086,Z 462.44,A -85,B 0,C 180,E1 13325.214,E2 13325.214} C_VEL
LIN {X 0,Y 332.579,Z 462.44,A -85,B 0,C 180,E1 13333.155,E2 13333.155} C_VEL
LIN {X 0,Y 332.298,Z 462.82,A -85,B 0,C 180,E1 13338.756,E2 13338.756} C_VEL
LIN {X 0,Y 334.044,Z 467.51,A -85,B 0,C 180,E1 13340.051,E2 13340.051} C_VEL
LIN {X 0,Y 338.071,Z 471.202,A -85,B 0,C 180,E1 13342.286,E2 13342.286} C_VEL
LIN {X 0,Y 342.068,Z 476.763,A -85,B 0,C 180,E1 13344.339,E2 13344.339} C_VEL
LIN {X 0,Y 349.806,Z 487.392,A -85,B 0,C 180,E1 13347.758,E2 13347.758} C_VEL
LIN {X 0,Y 361.977,Z 504.222,A -85,B 0,C 180,E1 13352.167,E2 13352.167} C_VEL
LIN {X 0,Y 377.889,Z 530.971,A -85,B 0,C 180,E1 13357.296,E2 13357.296} C_VEL
LIN {X 0,Y 391.331,Z 560.604,A -85,B 0,C 180,E1 13361.851,E2 13361.851} C_VEL
LIN {X 0,Y 391.675,Z 566.356,A -85,B 0,C 180,E1 13362.35,E2 13362.35} C_VEL
LIN {X 0,Y 383.823,Z 604.118,A -85,B 0,C 180,E1 13364.596,E2 13364.596} C_VEL
LIN {X 0,Y 374.505,Z 638.408,A -85,B 0,C 180,E1 13367.571,E2 13367.571} C_VEL
LIN {X 0,Y 364.342,Z 670.1,A -85,B 0,C 180,E1 13371.437,E2 13371.437} C_VEL
LIN {X 0,Y 354.295,Z 698.511,A -85,B 0,C 180,E1 13376.25,E2 13376.25} C_VEL
LIN {X 0,Y 345.512,Z 722.535,A -85,B 0,C 180,E1 13381.895,E2 13381.895} C_VEL
LIN {X 0,Y 339.167,Z 741.983,A -85,B 0,C 180,E1 13388.389,E2 13388.389} C_VEL
LIN {X 0,Y 335.505,Z 755.53,A -85,B 0,C 180,E1 13395.069,E2 13395.069} C_VEL
LIN {X 0,Y 334.14,Z 762.983,A -85,B 0,C 180,E1 13400.874,E2 13400.874} C_VEL
LIN {X 0,Y 333.579,Z 766.99,A -85,B 0,C 180,E1 13407.398,E2 13407.398} C_VEL
LIN {X 0,Y 333.577,Z 766.736,A -85,B 0,C 180,E1 13413.188,E2 13413.188} C_VEL
LIN {X 0,Y 334.153,Z 762.9,A -85,B 0,C 180,E1 13419.125,E2 13419.125} C_VEL
LIN {X 0,Y 336.062,Z 753.013,A -85,B 0,C 180,E1 13426.356,E2 13426.356} C_VEL
LIN {X 0,Y 340.21,Z 738.43,A -85,B 0,C 180,E1 13432.919,E2 13432.919} C_VEL
LIN {X 0,Y 347.288,Z 717.684,A -85,B 0,C 180,E1 13439.326,E2 13439.326} C_VEL
LIN {X 0,Y 356.756,Z 691.718,A -85,B 0,C 180,E1 13444.957,E2 13444.957} C_VEL
LIN {X 0,Y 366.886,Z 662.533,A -85,B 0,C 180,E1 13449.512,E2 13449.512} C_VEL
LIN {X 0,Y 377.047,Z 629.616,A -85,B 0,C 180,E1 13453.201,E2 13453.201} C_VEL
LIN {X 0,Y 386.233,Z 593.384,A -85,B 0,C 180,E1 13456.053,E2 13456.053} C_VEL
LIN {X 0,Y 391.876,Z 562.517,A -85,B 0,C 180,E1 13457.801,E2 13457.801} C_VEL
LIN {X 0,Y 379.255,Z 533.585,A -85,B 0,C 180,E1 13462.14,E2 13462.14} C_VEL
LIN {X 0,Y 364.112,Z 507.781,A -85,B 0,C 180,E1 13466.975,E2 13466.975} C_VEL
LIN {X 0,Y 351.509,Z 489.61,A -85,B 0,C 180,E1 13471.433,E2 13471.433} C_VEL
LIN {X 0,Y 346.289,Z 482.713,A -85,B 0,C 180,E1 13473.568,E2 13473.568} C_VEL
LIN {X 0,Y 341.769,Z 476.534,A -85,B 0,C 180,E1 13475.638,E2 13475.638} C_VEL
LIN {X 0,Y 337.97,Z 470.816,A -85,B 0,C 180,E1 13477.621,E2 13477.621} C_VEL
LIN {X 0,Y 332.671,Z 464.91,A -85,B 0,C 180,E1 13480.697,E2 13480.697} C_VEL
LIN {X 0,Y 332.317,Z 462.44,A -85,B 0,C 180,E1 13481.081,E2 13481.081} C_VEL
LIN {X 0,Y 332.683,Z 462.44,A -85,B 0,C 180,E1 13486.849,E2 13486.849} C_VEL
LIN {X 0,Y 333.156,Z 462.44,A -85,B 0,C 180,E1 13494.787,E2 13494.787} C_VEL
LIN {X 0,Y 333.396,Z 462.44,A -85,B 0,C 180,E1 13502.373,E2 13502.373} C_VEL
LIN {X 0,Y 332.72,Z 462.44,A -85,B 0,C 180,E1 13510.488,E2 13510.488} C_VEL
LIN {X 0,Y 332.474,Z 462.712,A -85,B 0,C 180,E1 13514.506,E2 13514.506} C_VEL
LIN {X 0,Y 334.336,Z 467.589,A -85,B 0,C 180,E1 13515.877,E2 13515.877} C_VEL
LIN {X 0,Y 338.172,Z 471.081,A -85,B 0,C 180,E1 13517.982,E2 13517.982} C_VEL
LIN {X 0,Y 342.359,Z 476.77,A -85,B 0,C 180,E1 13520.12,E2 13520.12} C_VEL
LIN {X 0,Y 353.65,Z 492.629,A -85,B 0,C 180,E1 13524.938,E2 13524.938} C_VEL
LIN {X 0,Y 368.289,Z 514.811,A -85,B 0,C 180,E1 13530.023,E2 13530.023} C_VEL
LIN {X 0,Y 382.665,Z 542.56,A -85,B 0,C 180,E1 13534.835,E2 13534.835} C_VEL
LIN {X 0,Y 391.786,Z 567.871,A -85,B 0,C 180,E1 13538.368,E2 13538.368} C_VEL
LIN {X 0,Y 383.749,Z 607.013,A -85,B 0,C 180,E1 13540.743,E2 13540.743} C_VEL
LIN {X 0,Y 374.681,Z 642.129,A -85,B 0,C 180,E1 13543.751,E2 13543.751} C_VEL
LIN {X 0,Y 364.063,Z 677.446,A -85,B 0,C 180,E1 13547.9,E2 13547.9} C_VEL
LIN {X 0,Y 354.259,Z 708.177,A -85,B 0,C 180,E1 13552.833,E2 13552.833} C_VEL
LIN {X 0,Y 345.712,Z 735.186,A -85,B 0,C 180,E1 13558.68,E2 13558.68} C_VEL
LIN {X 0,Y 339.614,Z 756.566,A -85,B 0,C 180,E1 13564.941,E2 13564.941} C_VEL
LIN {X 0,Y 335.57,Z 774.337,A -85,B 0,C 180,E1 13572.268,E2 13572.268} C_VEL
LIN {X 0,Y 333.885,Z 785.597,A -85,B 0,C 180,E1 13579.549,E2 13579.549} C_VEL
LIN {X 0,Y 333.559,Z 790.106,A -85,B 0,C 180,E1 13584.791,E2 13584.791} C_VEL
LIN {X 0,Y 333.677,Z 791.608,A -85,B 0,C 180,E1 13590,E2 13590} C_VEL
LIN {X 0,Y 333.555,Z 790.107,A -85,B 0,C 180,E1 13595.209,E2 13595.209} C_VEL
LIN {X 0,Y 334.063,Z 783.948,A -85,B 0,C 180,E1 13601.769,E2 13601.769} C_VEL
LIN {X 0,Y 335.819,Z 772.944,A -85,B 0,C 180,E1 13608.398,E2 13608.398} C_VEL
LIN {X 0,Y 338.533,Z 760.54,A -85,B 0,C 180,E1 13613.625,E2 13613.625} C_VEL
LIN {X 0,Y 336.662,Z 753.481,A -85,B 0,C 180,E1 13616.329,E2 13616.329} C_VEL
LIN {X 0,Y 335.17,Z 745.773,A -85,B 0,C 180,E1 13619.012,E2 13619.012} C_VEL
LIN {X 0,Y 343.281,Z 720.843,A -85,B 0,C 180,E1 13625.342,E2 13625.342} C_VEL
LIN {X 0,Y 353.273,Z 691.47,A -85,B 0,C 180,E1 13630.82,E2 13630.82} C_VEL
LIN {X 0,Y 364.13,Z 657.994,A -85,B 0,C 180,E1 13635.406,E2 13635.406} C_VEL
LIN {X 0,Y 374.669,Z 621.333,A -85,B 0,C 180,E1 13639.044,E2 13639.044} C_VEL
LIN {X 0,Y 383.972,Z 582.295,A -85,B 0,C 180,E1 13641.754,E2 13641.754} C_VEL
LIN {X 0,Y 385.949,Z 570.337,A -85,B 0,C 180,E1 13642.473,E2 13642.473} C_VEL
LIN {X 0,Y 376.838,Z 544.908,A -85,B 0,C 180,E1 13646.207,E2 13646.207} C_VEL
LIN {X 0,Y 363.983,Z 519.817,A -85,B 0,C 180,E1 13650.803,E2 13650.803} C_VEL
LIN {X 0,Y 349.701,Z 497.194,A -85,B 0,C 180,E1 13656.184,E2 13656.184} C_VEL
LIN {X 0,Y 339.615,Z 483.539,A -85,B 0,C 180,E1 13660.707,E2 13660.707} C_VEL
LIN {X 0,Y 334.909,Z 476.986,A -85,B 0,C 180,E1 13663.283,E2 13663.283} C_VEL
LIN {X 0,Y 330.758,Z 471.494,A -85,B 0,C 180,E1 13665.925,E2 13665.925} C_VEL
LIN {X 0,Y 329.671,Z 469.811,A -85,B 0,C 180,E1 13666.724,E2 13666.724} C_VEL
LIN {X 0,Y 325.274,Z 465.271,A -85,B 0,C 180,E1 13670.285,E2 13670.285} C_VEL
LIN {X 0,Y 324.848,Z 462.44,A -85,B 0,C 180,E1 13671.287,E2 13671.287} C_VEL
LIN {X 0,Y 325.451,Z 462.44,A -85,B 0,C 180,E1 13677.332,E2 13677.332} C_VEL
LIN {X 0,Y 325.372,Z 462.44,A -85,B 0,C 180,E1 13682.665,E2 13682.665} C_VEL
LIN {X 0,Y 324.775,Z 462.44,A -85,B 0,C 180,E1 13690.745,E2 13690.745} C_VEL
LIN {X 0,Y 324.674,Z 463.255,A -85,B 0,C 180,E1 13693.417,E2 13693.417} C_VEL
LIN {X 0,Y 326.631,Z 467.825,A -85,B 0,C 180,E1 13695.455,E2 13695.455} C_VEL
LIN {X 0,Y 330.544,Z 471.049,A -85,B 0,C 180,E1 13698.326,E2 13698.326} C_VEL
LIN {X 0,Y 333.919,Z 476.388,A -85,B 0,C 180,E1 13700.57,E2 13700.57} C_VEL
LIN {X 0,Y 336.256,Z 478.883,A -85,B 0,C 180,E1 13701.89,E2 13701.89} C_VEL
LIN {X 0,Y 342.588,Z 487.825,A -85,B 0,C 180,E1 13705.124,E2 13705.124} C_VEL
LIN {X 0,Y 351.081,Z 499.075,A -85,B 0,C 180,E1 13708.697,E2 13708.697} C_VEL
LIN {X 0,Y 365.334,Z 521.016,A -85,B 0,C 180,E1 13713.836,E2 13713.836} C_VEL
LIN {X 0,Y 378.879,Z 547.411,A -85,B 0,C 180,E1 13718.542,E2 13718.542} C_VEL
LIN {X 0,Y 386.539,Z 566.653,A -85,B 0,C 180,E1 13721.462,E2 13721.462} C_VEL
LIN {X 0,Y 378.741,Z 603.039,A -85,B 0,C 180,E1 13723.623,E2 13723.623} C_VEL
LIN {X 0,Y 369.099,Z 637.529,A -85,B 0,C 180,E1 13726.597,E2 13726.597} C_VEL
LIN {X 0,Y 358.77,Z 668.664,A -85,B 0,C 180,E1 13730.372,E2 13730.372} C_VEL
LIN {X 0,Y 348.198,Z 697.324,A -85,B 0,C 180,E1 13735.198,E2 13735.198} C_VEL
LIN {X 0,Y 338.801,Z 721.714,A -85,B 0,C 180,E1 13740.921,E2 13740.921} C_VEL
LIN {X 0,Y 332.14,Z 740.64,A -85,B 0,C 180,E1 13747.202,E2 13747.202} C_VEL
LIN {X 0,Y 328.092,Z 754.564,A -85,B 0,C 180,E1 13753.925,E2 13753.925} C_VEL
LIN {X 0,Y 326.283,Z 763.275,A -85,B 0,C 180,E1 13760.653,E2 13760.653} C_VEL
LIN {X 0,Y 325.695,Z 767.278,A -85,B 0,C 180,E1 13767.335,E2 13767.335} C_VEL
LIN {X 0,Y 325.745,Z 767.241,A -85,B 0,C 180,E1 13772.664,E2 13772.664} C_VEL
LIN {X 0,Y 326.297,Z 763.193,A -85,B 0,C 180,E1 13779.347,E2 13779.347} C_VEL
LIN {X 0,Y 328.376,Z 753.319,A -85,B 0,C 180,E1 13786.749,E2 13786.749} C_VEL
LIN {X 0,Y 332.777,Z 738.751,A -85,B 0,C 180,E1 13793.461,E2 13793.461} C_VEL
LIN {X 0,Y 340.289,Z 718.034,A -85,B 0,C 180,E1 13799.99,E2 13799.99} C_VEL
LIN {X 0,Y 350.202,Z 692.103,A -85,B 0,C 180,E1 13805.71,E2 13805.71} C_VEL
LIN {X 0,Y 361.031,Z 662.185,A -85,B 0,C 180,E1 13810.42,E2 13810.42} C_VEL
LIN {X 0,Y 371.66,Z 629.015,A -85,B 0,C 180,E1 13814.139,E2 13814.139} C_VEL
LIN {X 0,Y 380.678,Z 594.673,A -85,B 0,C 180,E1 13816.87,E2 13816.87} C_VEL
LIN {X 0,Y 386.337,Z 566.005,A -85,B 0,C 180,E1 13818.518,E2 13818.518} C_VEL
LIN {X 0,Y 374.548,Z 538.291,A -85,B 0,C 180,E1 13822.86,E2 13822.86} C_VEL
LIN {X 0,Y 360.347,Z 513.172,A -85,B 0,C 180,E1 13827.753,E2 13827.753} C_VEL
LIN {X 0,Y 348.105,Z 495.271,A -85,B 0,C 180,E1 13832.331,E2 13832.331} C_VEL
LIN {X 0,Y 339.639,Z 483.689,A -85,B 0,C 180,E1 13836.148,E2 13836.148} C_VEL
LIN {X 0,Y 334.75,Z 476.951,A -85,B 0,C 180,E1 13838.79,E2 13838.79} C_VEL
LIN {X 0,Y 330.686,Z 471.493,A -85,B 0,C 180,E1 13841.361,E2 13841.361} C_VEL
LIN {X 0,Y 329.416,Z 469.768,A -85,B 0,C 180,E1 13842.262,E2 13842.262} C_VEL
LIN {X 0,Y 325.058,Z 464.9,A -85,B 0,C 180,E1 13845.848,E2 13845.848} C_VEL
LIN {X 0,Y 324.739,Z 462.44,A -85,B 0,C 180,E1 13846.522,E2 13846.522} C_VEL
LIN {X 0,Y 325.226,Z 462.44,A -85,B 0,C 180,E1 13854.659,E2 13854.659} C_VEL
LIN {X 0,Y 325.596,Z 462.44,A -85,B 0,C 180,E1 13860.001,E2 13860.001} C_VEL
LIN {X 0,Y 325,Z 462.44,A -85,B 0,C 180,E1 13868.035,E2 13868.035} C_VEL
LIN {X 0,Y 324.876,Z 463.263,A -85,B 0,C 180,E1 13869.304,E2 13869.304} C_VEL
LIN {X 0,Y 327.491,Z 468.503,A -85,B 0,C 180,E1 13871.85,E2 13871.85} C_VEL
LIN {X 0,Y 330.761,Z 471.237,A -85,B 0,C 180,E1 13874.159,E2 13874.159} C_VEL
LIN {X 0,Y 334.613,Z 476.809,A -85,B 0,C 180,E1 13876.641,E2 13876.641} C_VEL
LIN {X 0,Y 336.62,Z 479.449,A -85,B 0,C 180,E1 13877.783,E2 13877.783} C_VEL
LIN {X 0,Y 342.389,Z 487.391,A -85,B 0,C 180,E1 13880.718,E2 13880.718} C_VEL
LIN {X 0,Y 351.332,Z 499.835,A -85,B 0,C 180,E1 13884.526,E2 13884.526} C_VEL
LIN {X 0,Y 365.199,Z 521.913,A -85,B 0,C 180,E1 13889.663,E2 13889.663} C_VEL
LIN {X 0,Y 378.557,Z 549.12,A -85,B 0,C 180,E1 13894.484,E2 13894.484} C_VEL
LIN {X 0,Y 385.882,Z 570.004,A -85,B 0,C 180,E1 13897.504,E2 13897.504} C_VEL
LIN {X 0,Y 376.985,Z 612.554,A -85,B 0,C 180,E1 13900.26,E2 13900.26} C_VEL
LIN {X 0,Y 366.585,Z 650.131,A -85,B 0,C 180,E1 13903.712,E2 13903.712} C_VEL
LIN {X 0,Y 355.404,Z 685.03,A -85,B 0,C 180,E1 13908.168,E2 13908.168} C_VEL
LIN {X 0,Y 344.935,Z 716.159,A -85,B 0,C 180,E1 13913.658,E2 13913.658} C_VEL
LIN {X 0,Y 336.449,Z 741.618,A -85,B 0,C 180,E1 13919.765,E2 13919.765} C_VEL
LIN {X 0,Y 330.261,Z 762.967,A -85,B 0,C 180,E1 13926.842,E2 13926.842} C_VEL
LIN {X 0,Y 327.115,Z 777.656,A -85,B 0,C 180,E1 13933.875,E2 13933.875} C_VEL
LIN {X 0,Y 325.884,Z 786.656,A -85,B 0,C 180,E1 13940.641,E2 13940.641} C_VEL
LIN {X 0,Y 325.735,Z 790.943,A -85,B 0,C 180,E1 13947.336,E2 13947.336} C_VEL
LIN {X 0,Y 325.657,Z 790.941,A -85,B 0,C 180,E1 13952.665,E2 13952.665} C_VEL
LIN {X 0,Y 325.909,Z 786.659,A -85,B 0,C 180,E1 13959.358,E2 13959.358} C_VEL
LIN {X 0,Y 327.126,Z 777.662,A -85,B 0,C 180,E1 13966.124,E2 13966.124} C_VEL
LIN {X 0,Y 330.29,Z 762.964,A -85,B 0,C 180,E1 13973.161,E2 13973.161} C_VEL
LIN {X 0,Y 335.17,Z 745.773,A -85,B 0,C 180,E1 13979.012,E2 13979.012} C_VEL
LIN {X 0,Y 334.208,Z 737.533,A -85,B 0,C 180,E1 13981.658,E2 13981.658} C_VEL
LIN {X 0,Y 333.594,Z 728.683,A -85,B 0,C 180,E1 13984.262,E2 13984.262} C_VEL
LIN {X 0,Y 343.694,Z 700.62,A -85,B 0,C 180,E1 13990.086,E2 13990.086} C_VEL
LIN {X 0,Y 354.741,Z 668.552,A -85,B 0,C 180,E1 13994.984,E2 13994.984} C_VEL
LIN {X 0,Y 365.724,Z 633.702,A -85,B 0,C 180,E1 13998.849,E2 13998.849} C_VEL
LIN {X 0,Y 375.715,Z 596.365,A -85,B 0,C 180,E1 14001.799,E2 14001.799} C_VEL
LIN {X 0,Y 380.165,Z 572.769,A -85,B 0,C 180,E1 14003.318,E2 14003.318} C_VEL
LIN {X 0,Y 371.195,Z 547.773,A -85,B 0,C 180,E1 14007.2,E2 14007.2} C_VEL
LIN {X 0,Y 358.955,Z 523.281,A -85,B 0,C 180,E1 14011.929,E2 14011.929} C_VEL
LIN {X 0,Y 346.574,Z 503.407,A -85,B 0,C 180,E1 14016.933,E2 14016.933} C_VEL
LIN {X 0,Y 337.474,Z 490.643,A -85,B 0,C 180,E1 14021.218,E2 14021.218} C_VEL
LIN {X 0,Y 332.859,Z 484.258,A -85,B 0,C 180,E1 14023.836,E2 14023.836} C_VEL
LIN {X 0,Y 328.76,Z 477.935,A -85,B 0,C 180,E1 14026.634,E2 14026.634} C_VEL
LIN {X 0,Y 323.873,Z 472.741,A -85,B 0,C 180,E1 14030.667,E2 14030.667} C_VEL
LIN {X 0,Y 322.864,Z 470.056,A -85,B 0,C 180,E1 14031.912,E2 14031.912} C_VEL
LIN {X 0,Y 318.42,Z 465.866,A -85,B 0,C 180,E1 14039.998,E2 14039.998} C_VEL
LIN {X 0,Y 319.164,Z 467.828,A -85,B 0,C 180,E1 14047.151,E2 14047.151} C_VEL
LIN {X 0,Y 323.239,Z 470.964,A -85,B 0,C 180,E1 14052.975,E2 14052.975} C_VEL
LIN {X 0,Y 326.102,Z 476.204,A -85,B 0,C 180,E1 14055.826,E2 14055.826} C_VEL
LIN {X 0,Y 328.928,Z 478.754,A -85,B 0,C 180,E1 14057.925,E2 14057.925} C_VEL
LIN {X 0,Y 333.299,Z 484.608,A -85,B 0,C 180,E1 14060.784,E2 14060.784} C_VEL
LIN {X 0,Y 344.458,Z 500.007,A -85,B 0,C 180,E1 14066.439,E2 14066.439} C_VEL
LIN {X 0,Y 357.39,Z 519.641,A -85,B 0,C 180,E1 14071.623,E2 14071.623} C_VEL
LIN {X 0,Y 370.742,Z 544.545,A -85,B 0,C 180,E1 14076.579,E2 14076.579} C_VEL
LIN {X 0,Y 380.715,Z 569.023,A -85,B 0,C 180,E1 14080.57,E2 14080.57} C_VEL
LIN {X 0,Y 372.113,Z 608.566,A -85,B 0,C 180,E1 14083.105,E2 14083.105} C_VEL
LIN {X 0,Y 361.683,Z 643.455,A -85,B 0,C 180,E1 14086.311,E2 14086.311} C_VEL
LIN {X 0,Y 350.072,Z 676.072,A -85,B 0,C 180,E1 14090.585,E2 14090.585} C_VEL
LIN {X 0,Y 339.434,Z 703.327,A -85,B 0,C 180,E1 14095.599,E2 14095.599} C_VEL
LIN {X 0,Y 330.041,Z 726.701,A -85,B 0,C 180,E1 14101.614,E2 14101.614} C_VEL
LIN {X 0,Y 323.266,Z 745.439,A -85,B 0,C 180,E1 14108.573,E2 14108.573} C_VEL
LIN {X 0,Y 319.818,Z 757.049,A -85,B 0,C 180,E1 14114.907,E2 14114.907} C_VEL
LIN {X 0,Y 318.2,Z 764.709,A -85,B 0,C 180,E1 14121.793,E2 14121.793} C_VEL
LIN {X 0,Y 317.815,Z 767.565,A -85,B 0,C 180,E1 14127.269,E2 14127.269} C_VEL
LIN {X 0,Y 317.846,Z 767.529,A -85,B 0,C 180,E1 14132.731,E2 14132.731} C_VEL
LIN {X 0,Y 318.45,Z 763.486,A -85,B 0,C 180,E1 14139.579,E2 14139.579} C_VEL
LIN {X 0,Y 320.714,Z 753.623,A -85,B 0,C 180,E1 14147.162,E2 14147.162} C_VEL
LIN {X 0,Y 325.39,Z 739.068,A -85,B 0,C 180,E1 14154.027,E2 14154.027} C_VEL
LIN {X 0,Y 333.401,Z 718.22,A -85,B 0,C 180,E1 14160.723,E2 14160.723} C_VEL
LIN {X 0,Y 343.708,Z 692.484,A -85,B 0,C 180,E1 14166.492,E2 14166.492} C_VEL
LIN {X 0,Y 354.602,Z 663.754,A -85,B 0,C 180,E1 14171.106,E2 14171.106} C_VEL
LIN {X 0,Y 365.795,Z 630.319,A -85,B 0,C 180,E1 14174.929,E2 14174.929} C_VEL
LIN {X 0,Y 375.523,Z 594.544,A -85,B 0,C 180,E1 14177.801,E2 14177.801} C_VEL
LIN {X 0,Y 380.9,Z 569.799,A -85,B 0,C 180,E1 14179.223,E2 14179.223} C_VEL
LIN {X 0,Y 369.362,Z 541.635,A -85,B 0,C 180,E1 14183.81,E2 14183.81} C_VEL
LIN {X 0,Y 355.06,Z 515.867,A -85,B 0,C 180,E1 14189.135,E2 14189.135} C_VEL
LIN {X 0,Y 342.472,Z 497.435,A -85,B 0,C 180,E1 14194.285,E2 14194.285} C_VEL
LIN {X 0,Y 336.734,Z 489.925,A -85,B 0,C 180,E1 14197.073,E2 14197.073} C_VEL
LIN {X 0,Y 332.729,Z 484.185,A -85,B 0,C 180,E1 14199.353,E2 14199.353} C_VEL
LIN {X 0,Y 328.804,Z 478.305,A -85,B 0,C 180,E1 14201.981,E2 14201.981} C_VEL
LIN {X 0,Y 323.612,Z 472.264,A -85,B 0,C 180,E1 14206.302,E2 14206.302} C_VEL
LIN {X 0,Y 322.766,Z 470.097,A -85,B 0,C 180,E1 14207.319,E2 14207.319} C_VEL
LIN {X 0,Y 318.054,Z 465.224,A -85,B 0,C 180,E1 14218.674,E2 14218.674} C_VEL
LIN {X 0,Y 323.384,Z 470.835,A -85,B 0,C 180,E1 14228.838,E2 14228.838} C_VEL
LIN {X 0,Y 326.673,Z 476.581,A -85,B 0,C 180,E1 14232.007,E2 14232.007} C_VEL
LIN {X 0,Y 329.118,Z 478.881,A -85,B 0,C 180,E1 14233.775,E2 14233.775} C_VEL
LIN {X 0,Y 333.652,Z 484.751,A -85,B 0,C 180,E1 14236.69,E2 14236.69} C_VEL
LIN {X 0,Y 344.803,Z 500.836,A -85,B 0,C 180,E1 14242.34,E2 14242.34} C_VEL
LIN {X 0,Y 356.248,Z 518.724,A -85,B 0,C 180,E1 14247.06,E2 14247.06} C_VEL
LIN {X 0,Y 369.253,Z 543.316,A -85,B 0,C 180,E1 14252.037,E2 14252.037} C_VEL
LIN {X 0,Y 379.469,Z 570.015,A -85,B 0,C 180,E1 14256.326,E2 14256.326} C_VEL
LIN {X 0,Y 380.035,Z 575.748,A -85,B 0,C 180,E1 14256.954,E2 14256.954} C_VEL
LIN {X 0,Y 370.809,Z 615.427,A -85,B 0,C 180,E1 14259.581,E2 14259.581} C_VEL
LIN {X 0,Y 360.344,Z 651.569,A -85,B 0,C 180,E1 14262.989,E2 14262.989} C_VEL
LIN {X 0,Y 348.828,Z 685.902,A -85,B 0,C 180,E1 14267.467,E2 14267.467} C_VEL
LIN {X 0,Y 337.737,Z 717.293,A -85,B 0,C 180,E1 14273.157,E2 14273.157} C_VEL
LIN {X 0,Y 328.712,Z 743.02,A -85,B 0,C 180,E1 14279.556,E2 14279.556} C_VEL
LIN {X 0,Y 322.647,Z 762.976,A -85,B 0,C 180,E1 14286.408,E2 14286.408} C_VEL
LIN {X 0,Y 319.329,Z 777.341,A -85,B 0,C 180,E1 14293.471,E2 14293.471} C_VEL
LIN {X 0,Y 317.993,Z 786.358,A -85,B 0,C 180,E1 14300.407,E2 14300.407} C_VEL
LIN {X 0,Y 317.844,Z 790.655,A -85,B 0,C 180,E1 14307.269,E2 14307.269} C_VEL
LIN {X 0,Y 317.751,Z 790.653,A -85,B 0,C 180,E1 14312.731,E2 14312.731} C_VEL
LIN {X 0,Y 318.018,Z 786.362,A -85,B 0,C 180,E1 14319.593,E2 14319.593} C_VEL
LIN {X 0,Y 319.338,Z 777.348,A -85,B 0,C 180,E1 14326.528,E2 14326.528} C_VEL
LIN {X 0,Y 322.668,Z 762.975,A -85,B 0,C 180,E1 14333.596,E2 14333.596} C_VEL
LIN {X 0,Y 329.242,Z 741.462,A -85,B 0,C 180,E1 14340.911,E2 14340.911} C_VEL
LIN {X 0,Y 333.594,Z 728.683,A -85,B 0,C 180,E1 14344.262,E2 14344.262} C_VEL
LIN {X 0,Y 333.501,Z 719.296,A -85,B 0,C 180,E1 14346.815,E2 14346.815} C_VEL
LIN {X 0,Y 333.922,Z 709.298,A -85,B 0,C 180,E1 14349.29,E2 14349.29} C_VEL
LIN {X 0,Y 345.439,Z 678.28,A -85,B 0,C 180,E1 14354.533,E2 14354.533} C_VEL
LIN {X 0,Y 356.775,Z 644.87,A -85,B 0,C 180,E1 14358.66,E2 14358.66} C_VEL
LIN {X 0,Y 367.354,Z 608.887,A -85,B 0,C 180,E1 14361.863,E2 14361.863} C_VEL
LIN {X 0,Y 374.79,Z 577.394,A -85,B 0,C 180,E1 14363.9,E2 14363.9} C_VEL
LIN {X 0,Y 367.198,Z 554.154,A -85,B 0,C 180,E1 14367.588,E2 14367.588} C_VEL
LIN {X 0,Y 355.336,Z 529.104,A -85,B 0,C 180,E1 14372.568,E2 14372.568} C_VEL
LIN {X 0,Y 343.526,Z 509.595,A -85,B 0,C 180,E1 14377.659,E2 14377.659} C_VEL
LIN {X 0,Y 335.149,Z 497.478,A -85,B 0,C 180,E1 14381.854,E2 14381.854} C_VEL
LIN {X 0,Y 330.834,Z 491.453,A -85,B 0,C 180,E1 14384.403,E2 14384.403} C_VEL
LIN {X 0,Y 326.315,Z 484.899,A -85,B 0,C 180,E1 14387.637,E2 14387.637} C_VEL
LIN {X 0,Y 322.247,Z 479.48,A -85,B 0,C 180,E1 14391.365,E2 14391.365} C_VEL
LIN {X 0,Y 320.977,Z 477.572,A -85,B 0,C 180,E1 14392.886,E2 14392.886} C_VEL
LIN {X 0,Y 317.456,Z 473.716,A -85,B 0,C 180,E1 14399.998,E2 14399.998} C_VEL
LIN {X 0,Y 318.211,Z 475.694,A -85,B 0,C 180,E1 14407.173,E2 14407.173} C_VEL
LIN {X 0,Y 321.929,Z 478.847,A -85,B 0,C 180,E1 14412.647,E2 14412.647} C_VEL
LIN {X 0,Y 325.596,Z 484.512,A -85,B 0,C 180,E1 14416.198,E2 14416.198} C_VEL
LIN {X 0,Y 327.614,Z 486.909,A -85,B 0,C 180,E1 14417.739,E2 14417.739} C_VEL
LIN {X 0,Y 333.225,Z 494.774,A -85,B 0,C 180,E1 14421.393,E2 14421.393} C_VEL
LIN {X 0,Y 342.215,Z 507.108,A -85,B 0,C 180,E1 14425.98,E2 14425.98} C_VEL
LIN {X 0,Y 354.288,Z 526.281,A -85,B 0,C 180,E1 14431.143,E2 14431.143} C_VEL
LIN {X 0,Y 366.675,Z 550.696,A -85,B 0,C 180,E1 14436.131,E2 14436.131} C_VEL
LIN {X 0,Y 375.204,Z 573.82,A -85,B 0,C 180,E1 14439.938,E2 14439.938} C_VEL
LIN {X 0,Y 366.174,Z 611.122,A -85,B 0,C 180,E1 14442.363,E2 14442.363} C_VEL
LIN {X 0,Y 355.517,Z 645.151,A -85,B 0,C 180,E1 14445.568,E2 14445.568} C_VEL
LIN {X 0,Y 343.591,Z 677.236,A -85,B 0,C 180,E1 14449.864,E2 14449.864} C_VEL
LIN {X 0,Y 332.276,Z 704.901,A -85,B 0,C 180,E1 14455.096,E2 14455.096} C_VEL
LIN {X 0,Y 322.442,Z 728.228,A -85,B 0,C 180,E1 14461.324,E2 14461.324} C_VEL
LIN {X 0,Y 315.428,Z 746.657,A -85,B 0,C 180,E1 14468.472,E2 14468.472} C_VEL
LIN {X 0,Y 311.606,Z 759.216,A -85,B 0,C 180,E1 14475.939,E2 14475.939} C_VEL
LIN {X 0,Y 310.335,Z 765,A -85,B 0,C 180,E1 14481.583,E2 14481.583} C_VEL
LIN {X 0,Y 309.914,Z 767.853,A -85,B 0,C 180,E1 14487.2,E2 14487.2} C_VEL
LIN {X 0,Y 309.944,Z 767.818,A -85,B 0,C 180,E1 14492.8,E2 14492.8} C_VEL
LIN {X 0,Y 310.602,Z 763.779,A -85,B 0,C 180,E1 14499.824,E2 14499.824} C_VEL
LIN {X 0,Y 313.046,Z 753.926,A -85,B 0,C 180,E1 14507.596,E2 14507.596} C_VEL
LIN {X 0,Y 318.018,Z 739.384,A -85,B 0,C 180,E1 14514.62,E2 14514.62} C_VEL
LIN {X 0,Y 326.508,Z 718.557,A -85,B 0,C 180,E1 14521.447,E2 14521.447} C_VEL
LIN {X 0,Y 337.269,Z 692.861,A -85,B 0,C 180,E1 14527.306,E2 14527.306} C_VEL
LIN {X 0,Y 348.905,Z 663.378,A -85,B 0,C 180,E1 14532.078,E2 14532.078} C_VEL
LIN {X 0,Y 360.206,Z 630.845,A -85,B 0,C 180,E1 14535.823,E2 14535.823} C_VEL
LIN {X 0,Y 370.558,Z 594.058,A -85,B 0,C 180,E1 14538.778,E2 14538.778} C_VEL
LIN {X 0,Y 375.137,Z 572.673,A -85,B 0,C 180,E1 14540.075,E2 14540.075} C_VEL
LIN {X 0,Y 364.379,Z 545.553,A -85,B 0,C 180,E1 14544.707,E2 14544.707} C_VEL
LIN {X 0,Y 351.309,Z 521.406,A -85,B 0,C 180,E1 14549.93,E2 14549.93} C_VEL
LIN {X 0,Y 340.224,Z 504.443,A -85,B 0,C 180,E1 14554.798,E2 14554.798} C_VEL
LIN {X 0,Y 331.017,Z 491.562,A -85,B 0,C 180,E1 14559.766,E2 14559.766} C_VEL
LIN {X 0,Y 325.976,Z 484.718,A -85,B 0,C 180,E1 14563.301,E2 14563.301} C_VEL
LIN {X 0,Y 321.999,Z 478.94,A -85,B 0,C 180,E1 14567.01,E2 14567.01} C_VEL
LIN {X 0,Y 317.069,Z 473.034,A -85,B 0,C 180,E1 14577.265,E2 14577.265} C_VEL
LIN {X 0,Y 318.088,Z 475.067,A -85,B 0,C 180,E1 14582.943,E2 14582.943} C_VEL
LIN {X 0,Y 322.087,Z 478.865,A -85,B 0,C 180,E1 14588.586,E2 14588.586} C_VEL
LIN {X 0,Y 325.863,Z 484.615,A -85,B 0,C 180,E1 14592.164,E2 14592.164} C_VEL
LIN {X 0,Y 327.792,Z 487.078,A -85,B 0,C 180,E1 14593.619,E2 14593.619} C_VEL
LIN {X 0,Y 333.265,Z 494.846,A -85,B 0,C 180,E1 14597.167,E2 14597.167} C_VEL
LIN {X 0,Y 341.684,Z 506.571,A -85,B 0,C 180,E1 14601.527,E2 14601.527} C_VEL
LIN {X 0,Y 354.738,Z 527.968,A -85,B 0,C 180,E1 14607.225,E2 14607.225} C_VEL
LIN {X 0,Y 366.605,Z 552.975,A -85,B 0,C 180,E1 14612.209,E2 14612.209} C_VEL
LIN {X 0,Y 374.759,Z 577.188,A -85,B 0,C 180,E1 14616.093,E2 14616.093} C_VEL
LIN {X 0,Y 365.402,Z 615.853,A -85,B 0,C 180,E1 14618.683,E2 14618.683} C_VEL
LIN {X 0,Y 354.462,Z 652.046,A -85,B 0,C 180,E1 14622.128,E2 14622.128} C_VEL
LIN {X 0,Y 342.44,Z 686.354,A -85,B 0,C 180,E1 14626.669,E2 14626.669} C_VEL
LIN {X 0,Y 331.105,Z 716.919,A -85,B 0,C 180,E1 14632.292,E2 14632.292} C_VEL
LIN {X 0,Y 321.64,Z 742.676,A -85,B 0,C 180,E1 14638.813,E2 14638.813} C_VEL
LIN {X 0,Y 315.055,Z 762.924,A -85,B 0,C 180,E1 14645.929,E2 14645.929} C_VEL
LIN {X 0,Y 311.364,Z 778.211,A -85,B 0,C 180,E1 14653.763,E2 14653.763} C_VEL
LIN {X 0,Y 310.107,Z 786.061,A -85,B 0,C 180,E1 14660.16,E2 14660.16} C_VEL
LIN {X 0,Y 309.934,Z 790.366,A -85,B 0,C 180,E1 14667.2,E2 14667.2} C_VEL
LIN {X 0,Y 309.845,Z 790.365,A -85,B 0,C 180,E1 14672.801,E2 14672.801} C_VEL
LIN {X 0,Y 310.131,Z 786.066,A -85,B 0,C 180,E1 14679.839,E2 14679.839} C_VEL
LIN {X 0,Y 311.582,Z 777.038,A -85,B 0,C 180,E1 14686.952,E2 14686.952} C_VEL
LIN {X 0,Y 315.07,Z 762.92,A -85,B 0,C 180,E1 14694.077,E2 14694.077} C_VEL
LIN {X 0,Y 322.013,Z 741.577,A -85,B 0,C 180,E1 14701.533,E2 14701.533} C_VEL
LIN {X 0,Y 331.738,Z 715.442,A -85,B 0,C 180,E1 14708.037,E2 14708.037} C_VEL
LIN {X 0,Y 333.922,Z 709.298,A -85,B 0,C 180,E1 14709.29,E2 14709.29} C_VEL
LIN {X 0,Y 334.788,Z 698.776,A -85,B 0,C 180,E1 14711.689,E2 14711.689} C_VEL
LIN {X 0,Y 335.936,Z 687.701,A -85,B 0,C 180,E1 14714.003,E2 14714.003} C_VEL
LIN {X 0,Y 347.752,Z 655.242,A -85,B 0,C 180,E1 14718.457,E2 14718.457} C_VEL
LIN {X 0,Y 359.231,Z 619.338,A -85,B 0,C 180,E1 14722.004,E2 14722.004} C_VEL
LIN {X 0,Y 369.209,Z 579.661,A -85,B 0,C 180,E1 14724.784,E2 14724.784} C_VEL
LIN {X 0,Y 360.097,Z 552.983,A -85,B 0,C 180,E1 14729.365,E2 14729.365} C_VEL
LIN {X 0,Y 348.043,Z 528.306,A -85,B 0,C 180,E1 14734.818,E2 14734.818} C_VEL
LIN {X 0,Y 337.461,Z 510.941,A -85,B 0,C 180,E1 14739.937,E2 14739.937} C_VEL
LIN {X 0,Y 329.219,Z 498.898,A -85,B 0,C 180,E1 14744.751,E2 14744.751} C_VEL
LIN {X 0,Y 324.501,Z 492.316,A -85,B 0,C 180,E1 14748.227,E2 14748.227} C_VEL
LIN {X 0,Y 320.697,Z 486.333,A -85,B 0,C 180,E1 14752.027,E2 14752.027} C_VEL
LIN {X 0,Y 316.487,Z 481.603,A -85,B 0,C 180,E1 14759.998,E2 14759.998} C_VEL
LIN {X 0,Y 317.112,Z 483.392,A -85,B 0,C 180,E1 14766.853,E2 14766.853} C_VEL
LIN {X 0,Y 320.674,Z 486.642,A -85,B 0,C 180,E1 14772.351,E2 14772.351} C_VEL
LIN {X 0,Y 324.681,Z 492.429,A -85,B 0,C 180,E1 14776.245,E2 14776.245} C_VEL
LIN {X 0,Y 331.573,Z 502.296,A -85,B 0,C 180,E1 14781.041,E2 14781.041} C_VEL
LIN {X 0,Y 340.412,Z 515.036,A -85,B 0,C 180,E1 14785.761,E2 14785.761} C_VEL
LIN {X 0,Y 352.059,Z 534.473,A -85,B 0,C 180,E1 14791.065,E2 14791.065} C_VEL
LIN {X 0,Y 363.488,Z 559.094,A -85,B 0,C 180,E1 14796.079,E2 14796.079} C_VEL
LIN {X 0,Y 369.715,Z 576.856,A -85,B 0,C 180,E1 14799.13,E2 14799.13} C_VEL
LIN {X 0,Y 360.337,Z 613.529,A -85,B 0,C 180,E1 14801.586,E2 14801.586} C_VEL
LIN {X 0,Y 349.432,Z 646.831,A -85,B 0,C 180,E1 14804.802,E2 14804.802} C_VEL
LIN {X 0,Y 337.247,Z 678.215,A -85,B 0,C 180,E1 14809.085,E2 14809.085} C_VEL
LIN {X 0,Y 325.709,Z 705.243,A -85,B 0,C 180,E1 14814.286,E2 14814.286} C_VEL
LIN {X 0,Y 315.86,Z 727.317,A -85,B 0,C 180,E1 14820.203,E2 14820.203} C_VEL
LIN {X 0,Y 308.729,Z 744.879,A -85,B 0,C 180,E1 14826.899,E2 14826.899} C_VEL
LIN {X 0,Y 304.361,Z 757.649,A -85,B 0,C 180,E1 14834.121,E2 14834.121} C_VEL
LIN {X 0,Y 302.472,Z 765.292,A -85,B 0,C 180,E1 14841.363,E2 14841.363} C_VEL
LIN {X 0,Y 302.012,Z 768.141,A -85,B 0,C 180,E1 14847.126,E2 14847.126} C_VEL
LIN {X 0,Y 302.041,Z 768.106,A -85,B 0,C 180,E1 14852.874,E2 14852.874} C_VEL
LIN {X 0,Y 302.748,Z 764.071,A -85,B 0,C 180,E1 14860.081,E2 14860.081} C_VEL
LIN {X 0,Y 305.037,Z 755.318,A -85,B 0,C 180,E1 14867.327,E2 14867.327} C_VEL
LIN {X 0,Y 310.03,Z 741.361,A -85,B 0,C 180,E1 14874.527,E2 14874.527} C_VEL
LIN {X 0,Y 318.566,Z 721.239,A -85,B 0,C 180,E1 14881.522,E2 14881.522} C_VEL
LIN {X 0,Y 329.511,Z 696.439,A -85,B 0,C 180,E1 14887.507,E2 14887.507} C_VEL
LIN {X 0,Y 341.632,Z 667.284,A -85,B 0,C 180,E1 14892.482,E2 14892.482} C_VEL
LIN {X 0,Y 353.781,Z 634.169,A -85,B 0,C 180,E1 14896.461,E2 14896.461} C_VEL
LIN {X 0,Y 365.022,Z 596.396,A -85,B 0,C 180,E1 14899.598,E2 14899.598} C_VEL
LIN {X 0,Y 369.501,Z 575.804,A -85,B 0,C 180,E1 14900.906,E2 14900.906} C_VEL
LIN {X 0,Y 359.051,Z 548.709,A -85,B 0,C 180,E1 14905.763,E2 14905.763} C_VEL
LIN {X 0,Y 346.109,Z 524.041,A -85,B 0,C 180,E1 14911.418,E2 14911.418} C_VEL
LIN {X 0,Y 334.349,Z 505.961,A -85,B 0,C 180,E1 14917.195,E2 14917.195} C_VEL
LIN {X 0,Y 328.513,Z 498.197,A -85,B 0,C 180,E1 14920.682,E2 14920.682} C_VEL
LIN {X 0,Y 324.624,Z 492.374,A -85,B 0,C 180,E1 14923.578,E2 14923.578} C_VEL
LIN {X 0,Y 320.607,Z 486.296,A -85,B 0,C 180,E1 14927.473,E2 14927.473} C_VEL
LIN {X 0,Y 316.103,Z 480.911,A -85,B 0,C 180,E1 14937.256,E2 14937.256} C_VEL
LIN {X 0,Y 317.172,Z 483.065,A -85,B 0,C 180,E1 14943.08,E2 14943.08} C_VEL
LIN {X 0,Y 320.797,Z 486.631,A -85,B 0,C 180,E1 14948.301,E2 14948.301} C_VEL
LIN {X 0,Y 324.895,Z 492.525,A -85,B 0,C 180,E1 14952.201,E2 14952.201} C_VEL
LIN {X 0,Y 331.589,Z 502.411,A -85,B 0,C 180,E1 14956.854,E2 14956.854} C_VEL
LIN {X 0,Y 340.089,Z 514.972,A -85,B 0,C 180,E1 14961.446,E2 14961.446} C_VEL
LIN {X 0,Y 351.622,Z 535.082,A -85,B 0,C 180,E1 14966.879,E2 14966.879} C_VEL
LIN {X 0,Y 362.466,Z 559.245,A -85,B 0,C 180,E1 14971.788,E2 14971.788} C_VEL
LIN {X 0,Y 369.16,Z 579.603,A -85,B 0,C 180,E1 14975.221,E2 14975.221} C_VEL
LIN {X 0,Y 359.214,Z 619.24,A -85,B 0,C 180,E1 14977.999,E2 14977.999} C_VEL
LIN {X 0,Y 348.387,Z 653.346,A -85,B 0,C 180,E1 14981.335,E2 14981.335} C_VEL
LIN {X 0,Y 336.399,Z 686.207,A -85,B 0,C 180,E1 14985.75,E2 14985.75} C_VEL
LIN {X 0,Y 324.586,Z 716.551,A -85,B 0,C 180,E1 14991.397,E2 14991.397} C_VEL
LIN {X 0,Y 314.612,Z 742.336,A -85,B 0,C 180,E1 14998.035,E2 14998.035} C_VEL
LIN {X 0,Y 307.59,Z 762.603,A -85,B 0,C 180,E1 15005.307,E2 15005.307} C_VEL
LIN {X 0,Y 303.578,Z 777.905,A -85,B 0,C 180,E1 15013.334,E2 15013.334} C_VEL
LIN {X 0,Y 302.234,Z 785.765,A -85,B 0,C 180,E1 15019.901,E2 15019.901} C_VEL
LIN {X 0,Y 302.023,Z 790.078,A -85,B 0,C 180,E1 15027.126,E2 15027.126} C_VEL
LIN {X 0,Y 301.953,Z 790.077,A -85,B 0,C 180,E1 15032.874,E2 15032.874} C_VEL
LIN {X 0,Y 302.255,Z 785.771,A -85,B 0,C 180,E1 15040.098,E2 15040.098} C_VEL
LIN {X 0,Y 303.815,Z 776.729,A -85,B 0,C 180,E1 15047.399,E2 15047.399} C_VEL
LIN {X 0,Y 307.585,Z 762.6,A -85,B 0,C 180,E1 15054.701,E2 15054.701} C_VEL
LIN {X 0,Y 314.988,Z 741.234,A -85,B 0,C 180,E1 15062.321,E2 15062.321} C_VEL
LIN {X 0,Y 325.255,Z 715.07,A -85,B 0,C 180,E1 15068.936,E2 15068.936} C_VEL
LIN {X 0,Y 335.936,Z 687.701,A -85,B 0,C 180,E1 15074.003,E2 15074.003} C_VEL
LIN {X 0,Y 337.268,Z 676.15,A -85,B 0,C 180,E1 15076.243,E2 15076.243} C_VEL
LIN {X 0,Y 338.418,Z 665.683,A -85,B 0,C 180,E1 15078.134,E2 15078.134} C_VEL
LIN {X 0,Y 339.006,Z 664.034,A -85,B 0,C 180,E1 15078.357,E2 15078.357} C_VEL
LIN {X 0,Y 351.635,Z 627.259,A -85,B 0,C 180,E1 15082.325,E2 15082.325} C_VEL
LIN {X 0,Y 363.175,Z 586.236,A -85,B 0,C 180,E1 15085.351,E2 15085.351} C_VEL
LIN {X 0,Y 363.574,Z 582.311,A -85,B 0,C 180,E1 15085.687,E2 15085.687} C_VEL
LIN {X 0,Y 355.328,Z 557.491,A -85,B 0,C 180,E1 15090.174,E2 15090.174} C_VEL
LIN {X 0,Y 344.562,Z 534.496,A -85,B 0,C 180,E1 15095.413,E2 15095.413} C_VEL
LIN {X 0,Y 334.733,Z 517.435,A -85,B 0,C 180,E1 15100.599,E2 15100.599} C_VEL
LIN {X 0,Y 327.132,Z 506.018,A -85,B 0,C 180,E1 15105.338,E2 15105.338} C_VEL
LIN {X 0,Y 323.131,Z 499.928,A -85,B 0,C 180,E1 15108.513,E2 15108.513} C_VEL
LIN {X 0,Y 319.31,Z 493.649,A -85,B 0,C 180,E1 15112.507,E2 15112.507} C_VEL
LIN {X 0,Y 315.52,Z 489.483,A -85,B 0,C 180,E1 15119.998,E2 15119.998} C_VEL
LIN {X 0,Y 316.152,Z 491.268,A -85,B 0,C 180,E1 15126.874,E2 15126.874} C_VEL
LIN {X 0,Y 319.433,Z 494.39,A -85,B 0,C 180,E1 15132.052,E2 15132.052} C_VEL
LIN {X 0,Y 323.764,Z 500.374,A -85,B 0,C 180,E1 15136.292,E2 15136.292} C_VEL
LIN {X 0,Y 330.764,Z 511.329,A -85,B 0,C 180,E1 15141.31,E2 15141.31} C_VEL
LIN {X 0,Y 340.458,Z 525.985,A -85,B 0,C 180,E1 15146.597,E2 15146.597} C_VEL
LIN {X 0,Y 351.522,Z 546.977,A -85,B 0,C 180,E1 15151.932,E2 15151.932} C_VEL
LIN {X 0,Y 361.548,Z 571.506,A -85,B 0,C 180,E1 15156.804,E2 15156.804} C_VEL
LIN {X 0,Y 364.18,Z 580.532,A -85,B 0,C 180,E1 15158.338,E2 15158.338} C_VEL
LIN {X 0,Y 353.695,Z 618.79,A -85,B 0,C 180,E1 15161.017,E2 15161.017} C_VEL
LIN {X 0,Y 341.578,Z 653.466,A -85,B 0,C 180,E1 15164.601,E2 15164.601} C_VEL
LIN {X 0,Y 328.509,Z 685.021,A -85,B 0,C 180,E1 15169.265,E2 15169.265} C_VEL
LIN {X 0,Y 316.302,Z 711.859,A -85,B 0,C 180,E1 15174.94,E2 15174.94} C_VEL
LIN {X 0,Y 306.637,Z 732.79,A -85,B 0,C 180,E1 15181.22,E2 15181.22} C_VEL
LIN {X 0,Y 299.61,Z 749.586,A -85,B 0,C 180,E1 15188.507,E2 15188.507} C_VEL
LIN {X 0,Y 295.656,Z 761.546,A -85,B 0,C 180,E1 15196.629,E2 15196.629} C_VEL
LIN {X 0,Y 294.207,Z 767.364,A -85,B 0,C 180,E1 15204.092,E2 15204.092} C_VEL
LIN {X 0,Y 294.237,Z 768.774,A -85,B 0,C 180,E1 15210,E2 15210} C_VEL
LIN {X 0,Y 294.212,Z 767.309,A -85,B 0,C 180,E1 15215.908,E2 15215.908} C_VEL
LIN {X 0,Y 295.7,Z 761.403,A -85,B 0,C 180,E1 15223.406,E2 15223.406} C_VEL
LIN {X 0,Y 299.64,Z 749.391,A -85,B 0,C 180,E1 15231.491,E2 15231.491} C_VEL
LIN {X 0,Y 307.189,Z 731.477,A -85,B 0,C 180,E1 15239.127,E2 15239.127} C_VEL
LIN {X 0,Y 317.059,Z 710.041,A -85,B 0,C 180,E1 15245.406,E2 15245.406} C_VEL
LIN {X 0,Y 329.245,Z 683.18,A -85,B 0,C 180,E1 15250.945,E2 15250.945} C_VEL
LIN {X 0,Y 341.639,Z 652.861,A -85,B 0,C 180,E1 15255.389,E2 15255.389} C_VEL
LIN {X 0,Y 353.849,Z 617.979,A -85,B 0,C 180,E1 15258.954,E2 15258.954} C_VEL
LIN {X 0,Y 364.005,Z 581.145,A -85,B 0,C 180,E1 15261.521,E2 15261.521} C_VEL
LIN {X 0,Y 358.734,Z 563.667,A -85,B 0,C 180,E1 15264.496,E2 15264.496} C_VEL
LIN {X 0,Y 347.252,Z 538.604,A -85,B 0,C 180,E1 15269.92,E2 15269.92} C_VEL
LIN {X 0,Y 336.166,Z 519.159,A -85,B 0,C 180,E1 15275.476,E2 15275.476} C_VEL
LIN {X 0,Y 327.05,Z 505.811,A -85,B 0,C 180,E1 15280.933,E2 15280.933} C_VEL
LIN {X 0,Y 322.86,Z 499.683,A -85,B 0,C 180,E1 15284.185,E2 15284.185} C_VEL
LIN {X 0,Y 318.592,Z 493.165,A -85,B 0,C 180,E1 15288.697,E2 15288.697} C_VEL
LIN {X 0,Y 315.159,Z 488.787,A -85,B 0,C 180,E1 15298.625,E2 15298.625} C_VEL
LIN {X 0,Y 319.505,Z 494.391,A -85,B 0,C 180,E1 15308.003,E2 15308.003} C_VEL
LIN {X 0,Y 323.805,Z 500.359,A -85,B 0,C 180,E1 15312.147,E2 15312.147} C_VEL
LIN {X 0,Y 333.181,Z 514.784,A -85,B 0,C 180,E1 15318.548,E2 15318.548} C_VEL
LIN {X 0,Y 343.713,Z 532.999,A -85,B 0,C 180,E1 15324.218,E2 15324.218} C_VEL
LIN {X 0,Y 354.705,Z 556.1,A -85,B 0,C 180,E1 15329.57,E2 15329.57} C_VEL
LIN {X 0,Y 363.17,Z 581.001,A -85,B 0,C 180,E1 15334.114,E2 15334.114} C_VEL
LIN {X 0,Y 363.371,Z 584.896,A -85,B 0,C 180,E1 15334.561,E2 15334.561} C_VEL
LIN {X 0,Y 352.048,Z 625.891,A -85,B 0,C 180,E1 15337.563,E2 15337.563} C_VEL
LIN {X 0,Y 339.118,Z 663.643,A -85,B 0,C 180,E1 15341.604,E2 15341.604} C_VEL
LIN {X 0,Y 326.61,Z 695.663,A -85,B 0,C 180,E1 15346.402,E2 15346.402} C_VEL
LIN {X 0,Y 314.615,Z 724.8,A -85,B 0,C 180,E1 15352.474,E2 15352.474} C_VEL
LIN {X 0,Y 304.579,Z 749.78,A -85,B 0,C 180,E1 15359.779,E2 15359.779} C_VEL
LIN {X 0,Y 298.133,Z 768.528,A -85,B 0,C 180,E1 15367.61,E2 15367.61} C_VEL
LIN {X 0,Y 295.201,Z 780.654,A -85,B 0,C 180,E1 15375.14,E2 15375.14} C_VEL
LIN {X 0,Y 294.225,Z 786.752,A -85,B 0,C 180,E1 15381.119,E2 15381.119} C_VEL
LIN {X 0,Y 294.112,Z 789.789,A -85,B 0,C 180,E1 15387.049,E2 15387.049} C_VEL
LIN {X 0,Y 294.045,Z 789.788,A -85,B 0,C 180,E1 15392.952,E2 15392.952} C_VEL
LIN {X 0,Y 294.394,Z 785.477,A -85,B 0,C 180,E1 15400.37,E2 15400.37} C_VEL
LIN {X 0,Y 296.078,Z 776.421,A -85,B 0,C 180,E1 15407.869,E2 15407.869} C_VEL
LIN {X 0,Y 300.3,Z 761.719,A -85,B 0,C 180,E1 15415.601,E2 15415.601} C_VEL
LIN {X 0,Y 308.484,Z 739.813,A -85,B 0,C 180,E1 15423.453,E2 15423.453} C_VEL
LIN {X 0,Y 319.111,Z 713.821,A -85,B 0,C 180,E1 15430.068,E2 15430.068} C_VEL
LIN {X 0,Y 331.608,Z 683.363,A -85,B 0,C 180,E1 15435.635,E2 15435.635} C_VEL
LIN {X 0,Y 339.006,Z 664.034,A -85,B 0,C 180,E1 15438.357,E2 15438.357} C_VEL
LIN {X 0,Y 340.958,Z 651.374,A -85,B 0,C 180,E1 15440.376,E2 15440.376} C_VEL
LIN {X 0,Y 342.914,Z 638.249,A -85,B 0,C 180,E1 15442.296,E2 15442.296} C_VEL
LIN {X 0,Y 355.117,Z 599.158,A -85,B 0,C 180,E1 15445.538,E2 15445.538} C_VEL
LIN {X 0,Y 358.329,Z 586.708,A -85,B 0,C 180,E1 15446.342,E2 15446.342} C_VEL
LIN {X 0,Y 350.989,Z 563.127,A -85,B 0,C 180,E1 15450.725,E2 15450.725} C_VEL
LIN {X 0,Y 340.808,Z 540.071,A -85,B 0,C 180,E1 15456.172,E2 15456.172} C_VEL
LIN {X 0,Y 331.097,Z 522.457,A -85,B 0,C 180,E1 15461.762,E2 15461.762} C_VEL
LIN {X 0,Y 324.933,Z 512.913,A -85,B 0,C 180,E1 15466.012,E2 15466.012} C_VEL
LIN {X 0,Y 321.42,Z 507.397,A -85,B 0,C 180,E1 15468.967,E2 15468.967} C_VEL
LIN {X 0,Y 317.519,Z 500.852,A -85,B 0,C 180,E1 15473.496,E2 15473.496} C_VEL
LIN {X 0,Y 314.553,Z 497.359,A -85,B 0,C 180,E1 15479.998,E2 15479.998} C_VEL
LIN {X 0,Y 315.063,Z 498.963,A -85,B 0,C 180,E1 15486.552,E2 15486.552} C_VEL
LIN {X 0,Y 318.202,Z 502.127,A -85,B 0,C 180,E1 15491.752,E2 15491.752} C_VEL
LIN {X 0,Y 323.297,Z 510.196,A -85,B 0,C 180,E1 15496.931,E2 15496.931} C_VEL
LIN {X 0,Y 330.839,Z 521.38,A -85,B 0,C 180,E1 15502.2,E2 15502.2} C_VEL
LIN {X 0,Y 341.387,Z 539.905,A -85,B 0,C 180,E1 15508.136,E2 15508.136} C_VEL
LIN {X 0,Y 352.058,Z 563.401,A -85,B 0,C 180,E1 15513.662,E2 15513.662} C_VEL
LIN {X 0,Y 358.566,Z 582.565,A -85,B 0,C 180,E1 15517.313,E2 15517.313} C_VEL
LIN {X 0,Y 348.544,Z 619.343,A -85,B 0,C 180,E1 15520.036,E2 15520.036} C_VEL
LIN {X 0,Y 336.026,Z 653.904,A -85,B 0,C 180,E1 15523.633,E2 15523.633} C_VEL
LIN {X 0,Y 322.254,Z 685.85,A -85,B 0,C 180,E1 15528.419,E2 15528.419} C_VEL
LIN {X 0,Y 309.081,Z 713.473,A -85,B 0,C 180,E1 15534.427,E2 15534.427} C_VEL
LIN {X 0,Y 298.672,Z 735.019,A -85,B 0,C 180,E1 15541.21,E2 15541.21} C_VEL
LIN {X 0,Y 291.584,Z 751.204,A -85,B 0,C 180,E1 15548.685,E2 15548.685} C_VEL
LIN {X 0,Y 287.864,Z 761.839,A -85,B 0,C 180,E1 15556.26,E2 15556.26} C_VEL
LIN {X 0,Y 286.319,Z 767.654,A -85,B 0,C 180,E1 15563.929,E2 15563.929} C_VEL
LIN {X 0,Y 286.365,Z 769.06,A -85,B 0,C 180,E1 15570,E2 15570} C_VEL
LIN {X 0,Y 286.325,Z 767.599,A -85,B 0,C 180,E1 15576.071,E2 15576.071} C_VEL
LIN {X 0,Y 287.906,Z 761.699,A -85,B 0,C 180,E1 15583.776,E2 15583.776} C_VEL
LIN {X 0,Y 292.128,Z 749.7,A -85,B 0,C 180,E1 15592.072,E2 15592.072} C_VEL
LIN {X 0,Y 300.121,Z 731.801,A -85,B 0,C 180,E1 15599.881,E2 15599.881} C_VEL
LIN {X 0,Y 310.766,Z 709.842,A -85,B 0,C 180,E1 15606.402,E2 15606.402} C_VEL
LIN {X 0,Y 323.207,Z 683.561,A -85,B 0,C 180,E1 15611.88,E2 15611.88} C_VEL
LIN {X 0,Y 336.586,Z 652.065,A -85,B 0,C 180,E1 15616.501,E2 15616.501} C_VEL
LIN {X 0,Y 348.703,Z 618.543,A -85,B 0,C 180,E1 15619.933,E2 15619.933} C_VEL
LIN {X 0,Y 358.658,Z 582.848,A -85,B 0,C 180,E1 15622.518,E2 15622.518} C_VEL
LIN {X 0,Y 350.031,Z 558.541,A -85,B 0,C 180,E1 15627.274,E2 15627.274} C_VEL
LIN {X 0,Y 339.298,Z 536.153,A -85,B 0,C 180,E1 15632.799,E2 15632.799} C_VEL
LIN {X 0,Y 329.885,Z 520.13,A -85,B 0,C 180,E1 15638.203,E2 15638.203} C_VEL
LIN {X 0,Y 324.069,Z 511.586,A -85,B 0,C 180,E1 15642.213,E2 15642.213} C_VEL
LIN {X 0,Y 321.312,Z 507.196,A -85,B 0,C 180,E1 15644.565,E2 15644.565} C_VEL
LIN {X 0,Y 317.38,Z 500.864,A -85,B 0,C 180,E1 15649.002,E2 15649.002} C_VEL
LIN {X 0,Y 314.196,Z 496.628,A -85,B 0,C 180,E1 15658.621,E2 15658.621} C_VEL
LIN {X 0,Y 318.211,Z 502.065,A -85,B 0,C 180,E1 15667.691,E2 15667.691} C_VEL
LIN {X 0,Y 323.243,Z 510.182,A -85,B 0,C 180,E1 15672.77,E2 15672.77} C_VEL
LIN {X 0,Y 330.615,Z 521.564,A -85,B 0,C 180,E1 15678.006,E2 15678.006} C_VEL
LIN {X 0,Y 340.416,Z 539.408,A -85,B 0,C 180,E1 15683.683,E2 15683.683} C_VEL
LIN {X 0,Y 350.148,Z 560.978,A -85,B 0,C 180,E1 15688.853,E2 15688.853} C_VEL
LIN {X 0,Y 357.875,Z 584.892,A -85,B 0,C 180,E1 15693.365,E2 15693.365} C_VEL
LIN {X 0,Y 357.642,Z 588.806,A -85,B 0,C 180,E1 15693.785,E2 15693.785} C_VEL
LIN {X 0,Y 346.292,Z 627.861,A -85,B 0,C 180,E1 15696.728,E2 15696.728} C_VEL
LIN {X 0,Y 333.434,Z 663.915,A -85,B 0,C 180,E1 15700.642,E2 15700.642} C_VEL
LIN {X 0,Y 319.881,Z 697.082,A -85,B 0,C 180,E1 15705.719,E2 15705.719} C_VEL
LIN {X 0,Y 307.549,Z 725.621,A -85,B 0,C 180,E1 15711.839,E2 15711.839} C_VEL
LIN {X 0,Y 297.418,Z 749.449,A -85,B 0,C 180,E1 15718.972,E2 15718.972} C_VEL
LIN {X 0,Y 290.545,Z 768.214,A -85,B 0,C 180,E1 15726.992,E2 15726.992} C_VEL
LIN {X 0,Y 287.389,Z 780.35,A -85,B 0,C 180,E1 15734.726,E2 15734.726} C_VEL
LIN {X 0,Y 286.342,Z 786.458,A -85,B 0,C 180,E1 15740.872,E2 15740.872} C_VEL
LIN {X 0,Y 286.208,Z 789.5,A -85,B 0,C 180,E1 15746.967,E2 15746.967} C_VEL
LIN {X 0,Y 286.153,Z 789.501,A -85,B 0,C 180,E1 15753.033,E2 15753.033} C_VEL
LIN {X 0,Y 286.514,Z 785.183,A -85,B 0,C 180,E1 15760.659,E2 15760.659} C_VEL
LIN {X 0,Y 288.358,Z 776.115,A -85,B 0,C 180,E1 15768.364,E2 15768.364} C_VEL
LIN {X 0,Y 292.717,Z 761.891,A -85,B 0,C 180,E1 15776.083,E2 15776.083} C_VEL
LIN {X 0,Y 301.161,Z 740.623,A -85,B 0,C 180,E1 15783.976,E2 15783.976} C_VEL
LIN {X 0,Y 312.535,Z 714.086,A -85,B 0,C 180,E1 15790.913,E2 15790.913} C_VEL
LIN {X 0,Y 325.89,Z 682.959,A -85,B 0,C 180,E1 15796.67,E2 15796.67} C_VEL
LIN {X 0,Y 339.668,Z 647.411,A -85,B 0,C 180,E1 15801.329,E2 15801.329} C_VEL
LIN {X 0,Y 342.914,Z 638.249,A -85,B 0,C 180,E1 15802.296,E2 15802.296} C_VEL
LIN {X 0,Y 345.132,Z 624.659,A -85,B 0,C 180,E1 15804.11,E2 15804.11} C_VEL
LIN {X 0,Y 347.053,Z 610.454,A -85,B 0,C 180,E1 15805.773,E2 15805.773} C_VEL
LIN {X 0,Y 352.707,Z 589.113,A -85,B 0,C 180,E1 15807.324,E2 15807.324} C_VEL
LIN {X 0,Y 345.3,Z 565.114,A -85,B 0,C 180,E1 15812.084,E2 15812.084} C_VEL
LIN {X 0,Y 335.75,Z 542.897,A -85,B 0,C 180,E1 15817.724,E2 15817.724} C_VEL
LIN {X 0,Y 327.102,Z 526.867,A -85,B 0,C 180,E1 15823.271,E2 15823.271} C_VEL
LIN {X 0,Y 320.076,Z 515.157,A -85,B 0,C 180,E1 15829.092,E2 15829.092} C_VEL
LIN {X 0,Y 315.886,Z 508.382,A -85,B 0,C 180,E1 15834.153,E2 15834.153} C_VEL
LIN {X 0,Y 313.513,Z 505.214,A -85,B 0,C 180,E1 15839.998,E2 15839.998} C_VEL
LIN {X 0,Y 314.007,Z 506.814,A -85,B 0,C 180,E1 15846.574,E2 15846.574} C_VEL
LIN {X 0,Y 316.846,Z 509.874,A -85,B 0,C 180,E1 15851.503,E2 15851.503} C_VEL
LIN {X 0,Y 321.792,Z 518.062,A -85,B 0,C 180,E1 15856.755,E2 15856.755} C_VEL
LIN {X 0,Y 328.647,Z 528.858,A -85,B 0,C 180,E1 15861.872,E2 15861.872} C_VEL
LIN {X 0,Y 338.311,Z 546.873,A -85,B 0,C 180,E1 15867.753,E2 15867.753} C_VEL
LIN {X 0,Y 347.68,Z 568.829,A -85,B 0,C 180,E1 15873.055,E2 15873.055} C_VEL
LIN {X 0,Y 353.148,Z 587.665,A -85,B 0,C 180,E1 15876.677,E2 15876.677} C_VEL
LIN {X 0,Y 341.844,Z 624.519,A -85,B 0,C 180,E1 15879.434,E2 15879.434} C_VEL
LIN {X 0,Y 329.312,Z 657.34,A -85,B 0,C 180,E1 15883.026,E2 15883.026} C_VEL
LIN {X 0,Y 315.446,Z 687.917,A -85,B 0,C 180,E1 15887.779,E2 15887.779} C_VEL
LIN {X 0,Y 302.527,Z 713.802,A -85,B 0,C 180,E1 15893.535,E2 15893.535} C_VEL
LIN {X 0,Y 291.59,Z 735.33,A -85,B 0,C 180,E1 15900.442,E2 15900.442} C_VEL
LIN {X 0,Y 284.09,Z 751.503,A -85,B 0,C 180,E1 15908.094,E2 15908.094} C_VEL
LIN {X 0,Y 280.078,Z 762.218,A -85,B 0,C 180,E1 15915.964,E2 15915.964} C_VEL
LIN {X 0,Y 278.433,Z 767.943,A -85,B 0,C 180,E1 15923.756,E2 15923.756} C_VEL
LIN {X 0,Y 278.466,Z 769.347,A -85,B 0,C 180,E1 15930,E2 15930} C_VEL
LIN {X 0,Y 278.438,Z 767.888,A -85,B 0,C 180,E1 15936.244,E2 15936.244} C_VEL
LIN {X 0,Y 280.152,Z 761.959,A -85,B 0,C 180,E1 15944.199,E2 15944.199} C_VEL
LIN {X 0,Y 284.659,Z 750.008,A -85,B 0,C 180,E1 15952.683,E2 15952.683} C_VEL
LIN {X 0,Y 293.131,Z 732.122,A -85,B 0,C 180,E1 15960.669,E2 15960.669} C_VEL
LIN {X 0,Y 304.181,Z 710.502,A -85,B 0,C 180,E1 15967.22,E2 15967.22} C_VEL
LIN {X 0,Y 317.279,Z 683.943,A -85,B 0,C 180,E1 15972.847,E2 15972.847} C_VEL
LIN {X 0,Y 331.111,Z 652.61,A -85,B 0,C 180,E1 15977.488,E2 15977.488} C_VEL
LIN {X 0,Y 344.188,Z 617.408,A -85,B 0,C 180,E1 15981.087,E2 15981.087} C_VEL
